C05352=1012.608,-74.665,-110.262,-31.652,71.658,-31.878
C05353=1012.607,-74.904,-110.243,-31.675,71.735,-31.896
C05354=1012.606,-75.144,-110.222,-31.698,71.811,-31.914
C05355=1012.605,-75.384,-110.202,-31.722,71.889,-31.932
C05356=1012.604,-75.624,-110.182,-31.745,71.965,-31.950
C05357=1012.603,-75.953,-110.153,-31.778,72.071,-31.977
C05358=1012.600,-76.343,-110.120,-31.818,72.198,-32.009
C05359=1012.601,-76.583,-110.100,-31.843,72.276,-32.028
C05360=1012.599,-76.822,-110.079,-31.869,72.354,-32.050
C05361=1012.598,-77.061,-110.059,-31.894,72.432,-32.070
C05362=1012.597,-77.300,-110.039,-31.920,72.510,-32.092
C05363=1012.596,-77.540,-110.019,-31.946,72.590,-32.112
C05364=1012.595,-77.779,-109.998,-31.973,72.668,-32.135
C05365=1012.594,-78.018,-109.978,-31.999,72.748,-32.156
C05366=1012.593,-78.257,-109.957,-32.027,72.828,-32.179
C05367=1012.593,-78.496,-109.937,-32.054,72.907,-32.201
C05368=1012.591,-78.734,-109.917,-32.082,72.987,-32.225
C05369=1012.591,-78.972,-109.897,-32.111,73.067,-32.250
C05370=1012.590,-79.211,-109.876,-32.140,73.147,-32.274
C05371=1012.588,-79.449,-109.856,-32.168,73.228,-32.298
C05372=1012.588,-79.687,-109.836,-32.198,73.307,-32.323
C05373=1012.587,-79.925,-109.816,-32.228,73.389,-32.349
C05374=1012.586,-80.163,-109.795,-32.257,73.470,-32.373
C05375=1012.585,-80.400,-109.775,-32.288,73.551,-32.400
C05376=1012.584,-80.637,-109.755,-32.318,73.632,-32.425
C05377=1012.583,-80.874,-109.735,-32.350,73.713,-32.453
C05378=1012.582,-81.111,-109.715,-32.382,73.795,-32.481
C05379=1012.581,-81.347,-109.694,-32.414,73.876,-32.509
C05380=1012.581,-81.583,-109.674,-32.446,73.958,-32.536
C05381=1012.579,-81.820,-109.654,-32.480,74.040,-32.567
C05382=1012.578,-82.058,-109.634,-32.514,74.123,-32.596
C05383=1012.578,-82.294,-109.614,-32.548,74.206,-32.626
C05384=1012.577,-82.532,-109.593,-32.582,74.288,-32.655
C05385=1012.576,-82.766,-109.574,-32.617,74.371,-32.686
C05386=1012.575,-83.003,-109.554,-32.651,74.454,-32.716
C05387=1012.574,-83.239,-109.533,-32.688,74.538,-32.750
C05388=1012.574,-83.475,-109.513,-32.724,74.621,-32.780
///RCONF 0,0,0,0,0,0,0,0,0,0,0,0,0,0,0,0,0,0,0,0,0,0,0,0
C05389=1012.572,-83.710,-109.494,-32.762,74.705,-32.815
C05390=1012.571,-83.943,-109.473,-32.799,74.787,-32.849
C05391=1012.570,-84.175,-109.454,-32.835,74.870,-32.879
C05392=1012.570,-84.409,-109.434,-32.874,74.953,-32.916
C05393=1012.568,-84.649,-109.413,-32.913,75.039,-32.951
C05394=1012.568,-84.904,-109.392,-32.956,75.132,-32.989
C05395=1012.568,-85.180,-109.368,-33.004,75.230,-33.034
C05396=1012.566,-85.465,-109.344,-33.054,75.334,-33.079
C05397=1012.565,-85.747,-109.320,-33.103,75.436,-33.124
C05398=1012.564,-86.017,-109.297,-33.153,75.535,-33.169
C05399=1012.563,-86.268,-109.276,-33.199,75.626,-33.211
C05400=1012.561,-86.502,-109.256,-33.242,75.712,-33.251
C05401=1012.561,-86.733,-109.236,-33.285,75.796,-33.290
C05402=1012.560,-86.963,-109.217,-33.331,75.881,-33.334
C05403=1012.560,-87.186,-109.198,-33.374,75.962,-33.374
C05404=1012.559,-87.405,-109.179,-33.418,76.044,-33.414
C05405=1012.558,-87.624,-109.160,-33.463,76.125,-33.455
C05406=1012.558,-87.840,-109.142,-33.506,76.204,-33.495
C05407=1012.556,-88.056,-109.123,-33.551,76.286,-33.538
C05408=1012.556,-88.282,-109.104,-33.600,76.369,-33.583
C05409=1012.555,-88.509,-109.084,-33.648,76.454,-33.628
C05410=1012.554,-88.742,-109.065,-33.700,76.541,-33.677
C05411=1012.553,-89.009,-109.042,-33.757,76.642,-33.730
C05412=1012.552,-89.306,-109.017,-33.825,76.753,-33.795
C05413=1012.552,-89.614,-108.991,-33.895,76.869,-33.860
C05414=1012.550,-89.915,-108.965,-33.967,76.983,-33.929
C05415=1012.549,-90.193,-108.942,-34.035,77.088,-33.993
C05416=1012.548,-90.433,-108.920,-34.094,77.180,-34.050
C05417=1012.547,-90.854,-108.885,-34.200,77.340,-34.150
C05418=1012.546,-91.137,-108.861,-34.274,77.448,-34.222
C05419=1012.545,-91.368,-108.841,-34.333,77.537,-34.278
C05420=1012.544,-91.600,-108.822,-34.396,77.626,-34.338
C05421=1012.543,-91.830,-108.802,-34.460,77.715,-34.400
C05422=1012.542,-92.061,-108.782,-34.525,77.804,-34.462
C05423=1012.542,-92.293,-108.763,-34.590,77.894,-34.525
C05424=1012.541,-92.523,-108.743,-34.657,77.983,-34.589
C05425=1012.541,-92.753,-108.723,-34.724,78.072,-34.654
C05426=1012.540,-92.983,-108.703,-34.792,78.162,-34.719
C05427=1012.539,-93.213,-108.683,-34.862,78.251,-34.787
C05428=1012.538,-93.443,-108.664,-34.935,78.341,-34.858
C05429=1012.538,-93.672,-108.645,-35.006,78.431,-34.927
C05430=1012.537,-93.901,-108.625,-35.080,78.520,-34.999
C05431=1012.536,-94.129,-108.606,-35.156,78.611,-35.072
C05432=1012.535,-94.357,-108.586,-35.232,78.700,-35.147
C05433=1012.535,-94.584,-108.567,-35.310,78.790,-35.223
C05434=1012.535,-94.811,-108.547,-35.388,78.880,-35.299
C05435=1012.534,-95.038,-108.529,-35.467,78.969,-35.376
C05436=1012.533,-95.265,-108.509,-35.551,79.059,-35.458
C05437=1012.532,-95.490,-108.490,-35.633,79.148,-35.538
C05438=1012.531,-95.716,-108.471,-35.719,79.238,-35.623
C05439=1012.530,-95.941,-108.451,-35.804,79.328,-35.706
C05440=1012.530,-96.166,-108.432,-35.893,79.418,-35.793
C05441=1012.530,-96.390,-108.413,-35.984,79.508,-35.883
C05442=1012.529,-96.614,-108.394,-36.074,79.597,-35.971
C05443=1012.528,-96.839,-108.375,-36.167,79.688,-36.062
C05444=1012.528,-97.063,-108.356,-36.263,79.777,-36.157
C05445=1012.527,-97.286,-108.337,-36.359,79.868,-36.252
C05446=1012.527,-97.510,-108.318,-36.459,79.958,-36.350
C05447=1012.526,-97.733,-108.299,-36.559,80.048,-36.449
C05448=1012.525,-97.957,-108.280,-36.662,80.139,-36.550
C05449=1012.525,-98.180,-108.261,-36.768,80.230,-36.656
C05450=1012.524,-98.405,-108.242,-36.875,80.320,-36.761
C05451=1012.524,-98.628,-108.223,-36.986,80.411,-36.872
C05452=1012.523,-98.852,-108.204,-37.099,80.503,-36.983
C05453=1012.522,-99.076,-108.185,-37.214,80.594,-37.097
C05454=1012.521,-99.300,-108.165,-37.332,80.685,-37.214
C05455=1012.521,-99.524,-108.146,-37.453,80.778,-37.334
C05456=1012.521,-99.749,-108.127,-37.575,80.869,-37.456
C05457=1012.520,-99.975,-108.108,-37.703,80.961,-37.583
C05458=1012.519,-100.200,-108.089,-37.833,81.054,-37.711
C05459=1012.518,-100.426,-108.070,-37.968,81.147,-37.846
C05460=1012.518,-100.652,-108.050,-38.106,81.241,-37.984
C05461=1012.517,-100.879,-108.032,-38.243,81.334,-38.120
C05462=1012.517,-101.106,-108.012,-38.390,81.428,-38.267
C05463=1012.517,-101.333,-107.993,-38.537,81.522,-38.413
C05464=1012.516,-101.561,-107.973,-38.691,81.616,-38.567
C05465=1012.515,-101.789,-107.954,-38.844,81.711,-38.718
C05466=1012.515,-102.018,-107.934,-39.008,81.806,-38.883
C05467=1012.515,-102.247,-107.915,-39.171,81.901,-39.046
C05468=1012.514,-102.476,-107.895,-39.339,81.996,-39.214
C05469=1012.513,-102.705,-107.876,-39.515,82.091,-39.389
C05470=1012.513,-102.934,-107.856,-39.694,82.188,-39.568
C05471=1012.513,-103.164,-107.837,-39.878,82.283,-39.753
C05472=1012.512,-103.394,-107.817,-40.070,82.379,-39.945
C05473=1012.512,-103.624,-107.797,-40.264,82.475,-40.138
C05474=1012.511,-103.940,-107.770,-40.542,82.608,-40.416
C05475=1012.510,-104.316,-107.739,-40.887,82.765,-40.762
C05476=1012.509,-104.546,-107.719,-41.106,82.862,-40.981
C05477=1012.509,-104.777,-107.699,-41.335,82.959,-41.211
C05478=1012.509,-105.008,-107.680,-41.567,83.055,-41.443
C05479=1012.508,-105.240,-107.660,-41.809,83.153,-41.685
C05480=1012.507,-105.471,-107.641,-42.059,83.250,-41.936
C05481=1012.507,-105.703,-107.621,-42.315,83.347,-42.193
C05482=1012.507,-105.934,-107.602,-42.580,83.445,-42.458
C05483=1012.506,-106.166,-107.581,-42.857,83.542,-42.736
C05484=1012.507,-106.400,-107.561,-43.142,83.641,-43.022
C05485=1012.505,-106.643,-107.541,-43.453,83.743,-43.334
C05486=1012.505,-106.896,-107.519,-43.783,83.849,-43.664
C05487=1012.505,-107.158,-107.497,-44.142,83.959,-44.025
C05488=1012.505,-107.428,-107.474,-44.528,84.074,-44.412
C05489=1012.504,-107.703,-107.451,-44.934,84.189,-44.819
C05490=1012.503,-107.980,-107.427,-45.362,84.305,-45.249
C05491=1012.503,-108.254,-107.404,-45.802,84.419,-45.692
C05492=1012.503,-108.523,-107.381,-46.257,84.532,-46.148
C05493=1012.503,-108.783,-107.359,-46.709,84.640,-46.601
C05494=1012.502,-109.033,-107.338,-47.169,84.745,-47.062
C05495=1012.502,-109.274,-107.318,-47.630,84.845,-47.525
C05496=1012.501,-109.507,-107.298,-48.097,84.942,-47.994
C05497=1012.501,-109.739,-107.278,-48.576,85.038,-48.475
C05498=1012.501,-109.970,-107.259,-49.075,85.134,-48.976
C05499=1012.501,-110.202,-107.239,-49.594,85.228,-49.497
C05500=1012.500,-110.434,-107.219,-50.135,85.324,-50.039
C05501=1012.500,-110.665,-107.199,-50.705,85.419,-50.612
C05502=1012.500,-110.897,-107.180,-51.293,85.513,-51.202
C05503=1012.499,-111.128,-107.160,-51.914,85.607,-51.825
C05504=1012.499,-111.359,-107.140,-52.563,85.700,-52.476
C05505=1012.499,-111.590,-107.121,-53.233,85.794,-53.148
C05506=1012.499,-111.822,-107.101,-53.942,85.886,-53.860
C05507=1012.498,-112.053,-107.082,-54.684,85.978,-54.605
C05508=1012.498,-112.284,-107.062,-55.462,86.070,-55.385
C05509=1012.499,-112.516,-107.042,-56.287,86.161,-56.212
C05510=1012.498,-112.748,-107.023,-57.142,86.251,-57.070
C05511=1012.498,-112.979,-107.003,-58.042,86.340,-57.972
C05512=1012.497,-113.210,-106.984,-58.994,86.429,-58.928
C05513=1012.498,-113.441,-106.964,-59.988,86.516,-59.924
C05514=1012.498,-113.672,-106.945,-61.044,86.603,-60.983
C05515=1012.498,-113.903,-106.925,-62.143,86.688,-62.085
C05516=1012.498,-114.135,-106.905,-63.313,86.772,-63.258
C05517=1012.497,-114.366,-106.886,-64.545,86.855,-64.493
C05518=1012.497,-114.598,-106.866,-65.843,86.936,-65.795
C05519=1012.496,-114.829,-106.846,-67.217,87.016,-67.172
C05520=1012.497,-115.061,-106.827,-68.666,87.095,-68.624
C05521=1012.497,-115.272,-106.810,-70.066,87.164,-70.028
C05522=1012.497,-115.485,-106.791,-71.544,87.233,-71.508
C05523=1012.497,-115.754,-106.768,-73.538,87.317,-73.507
C05524=1012.496,-115.985,-106.749,-75.331,87.386,-75.303
C05525=1012.496,-116.217,-106.729,-77.246,87.453,-77.222
C05526=1012.496,-116.447,-106.710,-79.234,87.516,-79.213
C05527=1012.496,-116.679,-106.690,-81.352,87.577,-81.336
C05528=1012.496,-116.910,-106.670,-83.577,87.635,-83.564
C05529=1012.496,-117.141,-106.651,-85.907,87.688,-85.899
C05530=1012.497,-117.373,-106.632,-88.359,87.738,-88.354
C05531=1012.497,-117.604,-106.612,-90.919,87.783,-90.919
C05532=1012.496,-117.835,-106.593,-93.576,87.824,-93.580
C05533=1012.497,-118.066,-106.573,-96.329,87.860,-96.336
C05534=1012.496,-118.297,-106.554,-99.188,87.891,-99.200
C05535=1012.496,-118.529,-106.534,-102.102,87.916,-102.119
C05536=1012.497,-118.759,-106.514,-105.100,87.936,-105.121
C05537=1012.496,-118.990,-106.495,-108.145,87.950,-108.171
C05538=1012.496,-119.222,-106.475,-111.225,87.958,-111.255
C05539=1012.497,-119.453,-106.456,-114.338,87.960,-114.373
C05540=1012.497,-119.684,-106.437,-117.448,87.956,-117.488
C05541=1012.497,-119.916,-106.417,-120.535,87.946,-120.579
C05542=1012.498,-120.147,-106.397,-123.598,87.930,-123.648
C05543=1012.497,-120.378,-106.378,-126.611,87.908,-126.666
C05544=1012.498,-120.608,-106.359,-129.528,87.881,-129.588
C05545=1012.498,-120.840,-106.339,-132.400,87.848,-132.465
C05546=1012.498,-121.070,-106.320,-135.162,87.810,-135.232
C05547=1012.498,-121.302,-106.300,-137.833,87.766,-137.910
C05548=1012.499,-121.533,-106.281,-140.407,87.718,-140.488
C05549=1012.498,-121.764,-106.262,-142.856,87.666,-142.943
C05550=1012.498,-121.996,-106.242,-145.213,87.609,-145.305
C05551=1012.499,-122.227,-106.222,-147.454,87.548,-147.552
C05552=1012.499,-122.457,-106.203,-149.582,87.484,-149.685
C05553=1012.499,-122.689,-106.184,-151.598,87.416,-151.707
C05554=1012.500,-122.920,-106.164,-153.513,87.344,-153.629
C05555=1012.499,-123.151,-106.145,-155.336,87.270,-155.458
C05556=1012.500,-123.382,-106.125,-157.042,87.194,-157.170
C05557=1012.500,-123.613,-106.105,-158.676,87.115,-158.810
C05558=1012.501,-123.844,-106.086,-160.231,87.033,-160.370
C05559=1012.500,-124.076,-106.067,-161.687,86.949,-161.833
C05560=1012.501,-124.306,-106.048,-163.063,86.863,-163.216
C05561=1012.502,-124.537,-106.028,-164.377,86.775,-164.537
C05562=1012.501,-124.768,-106.009,-165.619,86.686,-165.785
C05563=1012.502,-124.999,-105.989,-166.793,86.595,-166.966
C05564=1012.502,-125.230,-105.970,-167.904,86.502,-168.083
C05565=1012.503,-125.462,-105.950,-168.968,86.408,-169.154
C05566=1012.503,-125.692,-105.931,-169.965,86.313,-170.158
C05567=1012.503,-125.923,-105.912,-170.920,86.216,-171.120
C05568=1012.503,-126.155,-105.892,-171.826,86.118,-172.033
C05569=1012.504,-126.464,-105.867,-172.966,85.987,-173.183
C05570=1012.504,-126.848,-105.834,-174.287,85.819,-174.516
C05571=1012.505,-127.079,-105.815,-175.034,85.718,-175.270
C05572=1012.506,-127.309,-105.795,-175.744,85.615,-175.989
C05573=1012.507,-127.541,-105.776,-176.421,85.512,-176.672
C05574=1012.506,-127.772,-105.757,-177.074,85.407,-177.333
C05575=1012.507,-128.003,-105.737,-177.688,85.303,-177.955
C05576=1012.508,-128.233,-105.718,-178.282,85.198,-178.556
C05577=1012.509,-128.465,-105.699,-178.849,85.091,-179.131
C05578=1012.509,-128.695,-105.679,-179.390,84.985,-179.681
C05579=1012.509,-128.927,-105.660,-179.915,84.877,179.787
C05580=1012.509,-129.157,-105.640,179.584,84.768,179.277
C05581=1012.510,-129.389,-105.622,179.110,84.661,178.795
C05582=1012.511,-129.619,-105.602,178.644,84.551,178.321
C05583=1012.512,-129.850,-105.582,178.204,84.442,177.873
C05584=1012.513,-130.082,-105.564,177.783,84.332,177.442
C05585=1012.513,-130.312,-105.544,177.372,84.221,177.023
C05586=1012.513,-130.543,-105.525,176.979,84.110,176.621
C05587=1012.513,-130.774,-105.505,176.601,83.999,176.234
C05588=1012.514,-131.006,-105.486,176.233,83.886,175.858
C05589=1012.515,-131.236,-105.467,175.884,83.774,175.500
C05590=1012.516,-131.467,-105.447,175.545,83.661,175.151
C05591=1012.517,-131.698,-105.428,175.217,83.549,174.814
C05592=1012.517,-131.929,-105.409,174.903,83.435,174.491
C05593=1012.518,-132.160,-105.389,174.595,83.321,174.174
C05594=1012.518,-132.391,-105.371,174.299,83.207,173.869
C05595=1012.519,-132.622,-105.351,174.019,83.093,173.578
C05596=1012.520,-132.852,-105.332,173.739,82.978,173.290
C05597=1012.521,-133.084,-105.313,173.474,82.863,173.015
C05598=1012.521,-133.315,-105.293,173.220,82.747,172.750
C05599=1012.522,-133.545,-105.274,172.970,82.632,172.490
C05600=1012.523,-133.777,-105.255,172.728,82.516,172.238
C05601=1012.524,-134.007,-105.235,172.495,82.399,171.996
C05602=1012.845,-81.888,-107.547,164.895,61.170,160.790
C05603=1012.843,-81.675,-107.564,164.893,61.240,160.803
C05604=1012.841,-81.438,-107.584,164.892,61.318,160.818
C05605=1012.839,-81.201,-107.604,164.889,61.395,160.832
C05606=1012.837,-80.965,-107.625,164.887,61.471,160.846
C05607=1012.835,-80.729,-107.644,164.885,61.548,160.861
C05608=1012.834,-80.492,-107.664,164.883,61.625,160.875
C05609=1012.832,-80.255,-107.684,164.880,61.701,160.889
C05610=1012.830,-80.018,-107.704,164.880,61.777,160.904
C05611=1012.828,-79.779,-107.724,164.877,61.853,160.918
C05612=1012.827,-79.542,-107.744,164.875,61.929,160.933
C05613=1012.824,-79.303,-107.764,164.874,62.005,160.947
C05614=1012.823,-79.065,-107.784,164.872,62.081,160.962
C05615=1012.821,-78.827,-107.803,164.871,62.155,160.976
C05616=1012.819,-78.588,-107.823,164.870,62.230,160.991
C05617=1012.818,-78.349,-107.843,164.869,62.305,161.005
C05618=1012.816,-78.110,-107.864,164.867,62.380,161.019
C05619=1012.814,-77.871,-107.884,164.866,62.454,161.034
C05620=1012.813,-77.632,-107.904,164.865,62.528,161.048
C05621=1012.812,-77.393,-107.924,164.865,62.602,161.063
C05622=1012.809,-77.154,-107.944,164.863,62.676,161.077
C05623=1012.808,-76.914,-107.964,164.863,62.749,161.092
C05624=1012.807,-76.675,-107.984,164.861,62.822,161.106
C05625=1012.805,-76.435,-108.004,164.861,62.895,161.121
C05626=1012.803,-76.196,-108.025,164.860,62.968,161.135
C05627=1012.801,-75.956,-108.045,164.860,63.040,161.150
C05628=1012.800,-75.716,-108.065,164.859,63.112,161.164
C05629=1012.799,-75.476,-108.084,164.860,63.185,161.179
C05630=1012.797,-75.237,-108.105,164.859,63.256,161.193
C05631=1012.796,-74.996,-108.125,164.860,63.328,161.208
C05632=1012.794,-74.756,-108.145,164.859,63.399,161.222
C05633=1012.792,-74.517,-108.166,164.859,63.470,161.237
C05634=1012.791,-74.276,-108.186,164.859,63.541,161.251
C05635=1012.789,-74.036,-108.206,164.860,63.612,161.266
C05636=1012.788,-73.796,-108.227,164.860,63.681,161.280
C05637=1012.786,-73.556,-108.247,164.861,63.751,161.295
C05638=1012.785,-73.315,-108.267,164.860,63.821,161.309
C05639=1012.783,-73.075,-108.287,164.861,63.891,161.324
C05640=1012.782,-72.834,-108.307,164.862,63.960,161.338
C05641=1012.781,-72.594,-108.328,164.863,64.028,161.353
C05642=1012.779,-72.354,-108.348,164.864,64.098,161.368
C05643=1012.778,-72.113,-108.368,164.864,64.166,161.382
C05644=1012.776,-71.873,-108.388,164.865,64.235,161.396
C05645=1012.774,-71.633,-108.408,164.867,64.302,161.411
C05646=1012.773,-71.392,-108.428,164.868,64.370,161.426
C05647=1012.772,-71.151,-108.448,164.869,64.438,161.440
C05648=1012.771,-70.910,-108.469,164.870,64.505,161.454
C05649=1012.769,-70.670,-108.489,164.871,64.572,161.469
C05650=1012.768,-70.429,-108.509,164.873,64.639,161.483
C05651=1012.766,-70.188,-108.530,164.875,64.704,161.498
C05652=1012.765,-69.947,-108.550,164.875,64.771,161.512
C05653=1012.763,-69.706,-108.570,164.878,64.837,161.527
C05654=1012.762,-69.465,-108.591,164.879,64.902,161.541
C05655=1012.761,-69.225,-108.611,164.882,64.968,161.556
C05656=1012.760,-68.984,-108.631,164.883,65.032,161.570
C05657=1012.758,-68.743,-108.651,164.885,65.097,161.585
C05658=1012.757,-68.502,-108.671,164.886,65.162,161.599
C05659=1012.756,-68.262,-108.692,164.888,65.226,161.613
C05660=1012.754,-68.021,-108.712,164.891,65.290,161.628
C05661=1012.753,-67.780,-108.732,164.894,65.354,161.643
C05662=1012.752,-67.539,-108.752,164.896,65.417,161.657
C05663=1012.750,-67.299,-108.773,164.898,65.481,161.672
C05664=1012.749,-67.058,-108.793,164.900,65.543,161.686
C05665=1012.748,-66.818,-108.814,164.903,65.606,161.700
C05666=1012.746,-66.578,-108.834,164.905,65.668,161.714
C05667=1012.745,-66.337,-108.854,164.908,65.731,161.729
C05668=1012.744,-66.097,-108.875,164.910,65.792,161.743
C05669=1012.743,-65.856,-108.894,164.913,65.854,161.757
C05670=1012.742,-65.616,-108.914,164.916,65.915,161.772
C05671=1012.741,-65.376,-108.935,164.918,65.976,161.786
C05672=1012.739,-65.136,-108.955,164.921,66.036,161.800
C05673=1012.737,-64.754,-108.987,164.926,66.132,161.823
C05674=1012.736,-64.417,-109.015,164.931,66.216,161.843
C05675=1012.734,-64.178,-109.036,164.934,66.276,161.858
C05676=1012.734,-63.938,-109.056,164.938,66.335,161.872
C05677=1012.732,-63.699,-109.077,164.941,66.394,161.886
C05678=1012.731,-63.459,-109.097,164.943,66.453,161.900
C05679=1012.730,-63.221,-109.116,164.948,66.511,161.915
C05680=1012.729,-62.982,-109.136,164.951,66.569,161.929
C05681=1012.728,-62.743,-109.157,164.953,66.627,161.943
C05682=1012.726,-62.505,-109.177,164.958,66.684,161.957
C05683=1012.725,-62.266,-109.197,164.962,66.741,161.971
C05684=1012.724,-62.028,-109.217,164.965,66.798,161.985
C05685=1012.723,-61.790,-109.237,164.969,66.855,161.999
C05686=1012.723,-61.552,-109.257,164.973,66.911,162.014
C05687=1012.722,-61.314,-109.277,164.977,66.967,162.028
C05688=1012.720,-61.077,-109.297,164.980,67.023,162.041
C05689=1012.719,-60.840,-109.317,164.984,67.078,162.056
C05690=1012.718,-60.603,-109.337,164.987,67.133,162.069
C05691=1012.717,-60.365,-109.356,164.992,67.187,162.083
C05692=1012.716,-60.129,-109.377,164.996,67.242,162.097
C05693=1012.715,-59.892,-109.396,165.001,67.296,162.111
C05694=1012.714,-59.656,-109.417,165.005,67.350,162.125
C05695=1012.713,-59.420,-109.437,165.009,67.403,162.139
C05696=1012.712,-59.183,-109.457,165.013,67.457,162.153
C05697=1012.710,-58.948,-109.476,165.018,67.510,162.167
C05698=1012.710,-58.711,-109.496,165.022,67.562,162.181
C05699=1012.710,-58.477,-109.516,165.027,67.615,162.195
C05700=1012.708,-58.242,-109.536,165.031,67.666,162.208
C05701=1012.707,-58.006,-109.556,165.036,67.719,162.222
C05702=1012.706,-57.771,-109.576,165.040,67.770,162.236
C05703=1012.705,-57.536,-109.595,165.045,67.821,162.250
C05704=1012.704,-57.302,-109.615,165.049,67.872,162.263
C05705=1012.704,-57.068,-109.635,165.053,67.923,162.276
C05706=1012.702,-56.833,-109.654,165.058,67.973,162.290
C05707=1012.701,-56.599,-109.674,165.063,68.023,162.304
C05708=1012.701,-56.365,-109.694,165.069,68.073,162.318
C05709=1012.699,-56.131,-109.714,165.073,68.123,162.331
C05710=1012.698,-55.897,-109.733,165.078,68.172,162.345
C05711=1012.697,-55.663,-109.753,165.084,68.221,162.358
C05712=1012.697,-55.429,-109.773,165.088,68.269,162.371
C05713=1012.697,-55.196,-109.793,165.092,68.318,162.385
C05714=1012.695,-54.962,-109.813,165.098,68.367,162.399
C05715=1012.694,-54.728,-109.832,165.103,68.414,162.412
C05716=1012.693,-54.494,-109.852,165.108,68.463,162.425
C05717=1012.693,-54.261,-109.871,165.113,68.510,162.438
C05718=1012.692,-54.027,-109.891,165.118,68.557,162.452
C05719=1012.691,-53.794,-109.911,165.123,68.604,162.465
C05720=1012.690,-53.560,-109.930,165.128,68.651,162.479
C05721=1012.689,-53.326,-109.950,165.134,68.697,162.492
C05722=1012.688,-53.092,-109.970,165.139,68.745,162.505
C05723=1012.687,-52.858,-109.989,165.145,68.791,162.519
C05724=1012.686,-52.625,-110.009,165.150,68.836,162.532
C05725=1012.686,-52.392,-110.029,165.156,68.882,162.545
C05726=1012.685,-52.157,-110.049,165.161,68.927,162.558
C05727=1012.685,-51.923,-110.068,165.166,68.972,162.571
C05728=1012.683,-51.689,-110.088,165.172,69.017,162.584
C05729=1012.682,-51.456,-110.108,165.177,69.062,162.598
C05730=1012.681,-51.222,-110.127,165.182,69.106,162.610
C05731=1012.681,-50.989,-110.147,165.189,69.151,162.624
C05732=1012.680,-50.755,-110.167,165.194,69.195,162.637
C05733=1012.680,-50.521,-110.187,165.200,69.237,162.650
C05734=1012.679,-50.287,-110.206,165.206,69.281,162.663
C05735=1012.678,-50.053,-110.226,165.212,69.324,162.676
C05736=1012.677,-49.819,-110.245,165.217,69.368,162.689
C05737=1012.677,-49.586,-110.265,165.222,69.410,162.702
C05738=1012.675,-49.352,-110.285,165.228,69.453,162.715
C05739=1012.675,-49.118,-110.305,165.235,69.496,162.728
C05740=1012.674,-48.884,-110.325,165.241,69.537,162.741
C05741=1012.673,-48.650,-110.344,165.246,69.579,162.754
C05742=1012.672,-48.416,-110.364,165.253,69.620,162.767
C05743=1012.672,-48.183,-110.383,165.259,69.662,162.780
C05744=1012.672,-47.949,-110.404,165.265,69.703,162.792
C05745=1012.671,-47.715,-110.423,165.270,69.743,162.805
C05746=1012.670,-47.481,-110.442,165.276,69.784,162.817
C05747=1012.669,-47.248,-110.462,165.281,69.825,162.830
C05748=1012.669,-47.013,-110.482,165.288,69.865,162.843
C05749=1012.667,-46.779,-110.502,165.294,69.904,162.856
C05750=1012.666,-46.545,-110.521,165.300,69.944,162.868
C05751=1012.666,-46.312,-110.541,165.306,69.983,162.881
C05752=1012.666,-46.078,-110.561,165.312,70.023,162.893
C05753=1012.665,-45.844,-110.581,165.319,70.062,162.906
C05754=1012.664,-45.610,-110.600,165.325,70.100,162.918
C05755=1012.664,-45.376,-110.620,165.330,70.139,162.930
C05756=1012.663,-45.142,-110.640,165.336,70.177,162.943
C05757=1012.662,-44.908,-110.659,165.343,70.215,162.955
C05758=1012.662,-44.674,-110.679,165.348,70.253,162.967
C05759=1012.661,-44.440,-110.698,165.356,70.290,162.980
C05760=1012.661,-44.206,-110.718,165.362,70.328,162.992
C05761=1012.659,-43.972,-110.739,165.368,70.365,163.005
C05762=1012.659,-43.739,-110.758,165.375,70.402,163.017
C05763=1012.658,-43.504,-110.778,165.380,70.438,163.029
C05764=1012.658,-43.270,-110.798,165.385,70.474,163.040
C05765=1012.657,-43.036,-110.817,165.394,70.511,163.054
C05766=1012.656,-42.802,-110.837,165.400,70.547,163.065
C05767=1012.656,-42.569,-110.856,165.406,70.582,163.077
C05768=1012.655,-42.334,-110.876,165.412,70.618,163.089
C05769=1012.655,-42.100,-110.896,165.418,70.653,163.101
C05770=1012.654,-41.866,-110.916,165.424,70.687,163.113
C05771=1012.653,-41.632,-110.935,165.430,70.722,163.124
C05772=1012.653,-41.397,-110.955,165.437,70.756,163.137
C05773=1012.652,-41.164,-110.975,165.444,70.791,163.149
C05774=1012.651,-40.929,-110.995,165.450,70.825,163.160
C05775=1012.651,-40.695,-111.014,165.456,70.858,163.172
C05776=1012.650,-40.461,-111.034,165.461,70.892,163.183
C05777=1012.650,-40.227,-111.054,165.469,70.925,163.195
C05778=1012.649,-39.993,-111.073,165.476,70.959,163.207
C05779=1012.649,-39.758,-111.093,165.481,70.992,163.218
C05780=1012.647,-39.380,-111.125,165.492,71.044,163.237
C05781=1012.647,-39.056,-111.152,165.500,71.089,163.252
C05782=1012.646,-38.822,-111.172,165.506,71.121,163.264
C05783=1012.646,-38.587,-111.192,165.512,71.152,163.275
C05784=1012.645,-38.353,-111.212,165.520,71.184,163.287
C05785=1012.645,-38.119,-111.231,165.526,71.216,163.298
C05786=1012.644,-37.885,-111.251,165.533,71.246,163.309
C05787=1012.644,-37.651,-111.271,165.538,71.277,163.320
C05788=1012.644,-37.416,-111.291,165.545,71.307,163.331
C05789=1012.643,-37.183,-111.310,165.551,71.338,163.342
C05790=1012.642,-36.948,-111.330,165.557,71.368,163.353
C05791=1012.642,-36.714,-111.350,165.563,71.398,163.363
C05792=1012.641,-36.480,-111.369,165.570,71.427,163.375
C05793=1012.640,-36.245,-111.390,165.577,71.457,163.386
C05794=1012.640,-36.011,-111.409,165.583,71.486,163.396
C05795=1012.639,-35.777,-111.429,165.589,71.515,163.407
C05796=1012.639,-35.543,-111.449,165.595,71.543,163.417
C05797=1012.639,-35.308,-111.468,165.601,71.572,163.428
C05798=1012.638,-35.074,-111.487,165.608,71.600,163.439
C05799=1012.637,-34.839,-111.507,165.613,71.629,163.449
C05800=1012.637,-34.605,-111.527,165.620,71.657,163.460
C05801=1012.636,-34.371,-111.546,165.626,71.684,163.470
C05802=1012.636,-34.137,-111.566,165.632,71.712,163.481
C05803=1012.636,-33.902,-111.586,165.638,71.738,163.491
C05804=1012.635,-33.668,-111.606,165.644,71.765,163.501
C05805=1012.635,-33.434,-111.625,165.650,71.791,163.511
C05806=1012.635,-33.200,-111.645,165.657,71.819,163.522
C05807=1012.634,-32.965,-111.666,165.663,71.845,163.532
C05808=1012.633,-32.731,-111.685,165.668,71.871,163.541
C05809=1012.632,-32.497,-111.705,165.674,71.897,163.551
C05810=1012.632,-32.262,-111.725,165.681,71.922,163.562
C05811=1012.631,-32.028,-111.744,165.686,71.948,163.571
C05812=1012.631,-31.794,-111.764,165.693,71.972,163.581
C05813=1012.631,-31.560,-111.784,165.699,71.997,163.591
C05814=1012.631,-31.325,-111.804,165.705,72.022,163.600
C05815=1012.630,-31.091,-111.823,165.710,72.046,163.609
C05816=1012.630,-30.857,-111.843,165.716,72.071,163.619
C05817=1012.629,-30.622,-111.863,165.723,72.094,163.629
C05818=1012.629,-30.389,-111.882,165.728,72.118,163.638
C05819=1012.628,-30.154,-111.902,165.734,72.142,163.647
C05820=1012.628,-29.920,-111.922,165.740,72.165,163.657
C05821=1012.628,-29.685,-111.942,165.745,72.188,163.666
C05822=1012.627,-29.452,-111.961,165.751,72.211,163.675
C05823=1012.627,-29.217,-111.981,165.758,72.234,163.684
C05824=1012.626,-28.982,-112.000,165.763,72.256,163.693
C05825=1012.625,-28.748,-112.020,165.769,72.278,163.702
C05826=1012.625,-28.514,-112.040,165.775,72.300,163.712
C05827=1012.625,-28.279,-112.059,165.780,72.322,163.720
C05828=1012.625,-28.045,-112.079,165.785,72.343,163.728
C05829=1012.624,-27.811,-112.099,165.792,72.365,163.738
C05830=1012.624,-27.577,-112.119,165.798,72.386,163.747
C05831=1012.623,-27.342,-112.138,165.801,72.407,163.754
C05832=1012.622,-27.109,-112.158,165.808,72.427,163.763
C05833=1012.622,-26.874,-112.178,165.813,72.447,163.771
C05834=1012.622,-26.640,-112.198,165.819,72.468,163.780
C05835=1012.621,-26.407,-112.218,165.824,72.488,163.788
C05836=1012.621,-26.172,-112.238,165.829,72.508,163.796
C05837=1012.621,-25.938,-112.257,165.835,72.527,163.805
C05838=1012.621,-25.703,-112.277,165.840,72.546,163.812
C05839=1012.620,-25.469,-112.297,165.845,72.566,163.820
C05840=1012.620,-25.235,-112.317,165.851,72.584,163.829
C05841=1012.619,-25.001,-112.336,165.856,72.603,163.836
C05842=1012.619,-24.767,-112.355,165.860,72.621,163.844
C05843=1012.619,-24.533,-112.375,165.865,72.640,163.852
C05844=1012.619,-24.298,-112.395,165.870,72.657,163.859
C05845=1012.618,-24.064,-112.414,165.876,72.675,163.867
C05846=1012.618,-23.830,-112.434,165.881,72.693,163.874
C05847=1012.618,-23.596,-112.454,165.885,72.710,163.882
C05848=1012.617,-23.362,-112.473,165.890,72.727,163.889
C05849=1012.616,-23.127,-112.493,165.895,72.744,163.896
C05850=1012.616,-22.893,-112.513,165.901,72.761,163.904
C05851=1012.615,-22.659,-112.533,165.906,72.777,163.911
C05852=1012.615,-22.425,-112.552,165.909,72.793,163.917
C05853=1012.615,-22.190,-112.572,165.913,72.809,163.924
C05854=1012.615,-21.958,-112.592,165.918,72.825,163.931
C05855=1012.615,-21.723,-112.612,165.924,72.841,163.938
C05856=1012.615,-21.489,-112.632,165.928,72.856,163.945
C05857=1012.614,-21.255,-112.651,165.933,72.871,163.951
C05858=1012.614,-21.020,-112.671,165.939,72.886,163.959
C05859=1012.613,-20.786,-112.691,165.942,72.901,163.965
C05860=1012.612,-20.552,-112.710,165.946,72.916,163.971
C05861=1012.612,-20.318,-112.730,165.950,72.929,163.977
C05862=1012.612,-20.040,-112.753,165.955,72.946,163.984
C05863=1012.612,-19.690,-112.783,165.963,72.967,163.994
C05864=1012.611,-19.430,-112.805,165.967,72.982,164.001
C05865=1012.611,-19.130,-112.830,165.972,72.999,164.008
C05866=1012.611,-18.804,-112.857,165.977,73.016,164.016
C05867=1012.610,-18.472,-112.885,165.984,73.035,164.024
C05868=1012.609,-18.155,-112.911,165.989,73.052,164.032
C05869=1012.610,-17.870,-112.936,165.994,73.066,164.039
C05870=1012.609,-17.623,-112.956,165.997,73.079,164.044
C05871=1012.609,-17.392,-112.976,166.002,73.090,164.050
C05872=1012.609,-17.161,-112.995,166.006,73.102,164.055
C05873=1012.609,-16.927,-113.015,166.008,73.113,164.059
C05874=1012.608,-16.689,-113.035,166.014,73.124,164.065
C05875=1012.608,-16.452,-113.055,166.016,73.135,164.070
C05876=1012.607,-16.217,-113.075,166.020,73.145,164.075
C05877=1012.607,-15.981,-113.094,166.024,73.156,164.080
C05878=1012.606,-15.745,-113.115,166.027,73.166,164.085
C05879=1012.606,-15.509,-113.134,166.030,73.176,164.089
C05880=1012.606,-15.277,-113.154,166.033,73.186,164.094
C05881=1012.605,-15.047,-113.173,166.037,73.195,164.098
C05882=1012.606,-14.820,-113.193,166.040,73.204,164.103
C05883=1012.605,-14.595,-113.211,166.042,73.213,164.106
C05884=1012.605,-14.372,-113.230,166.046,73.222,164.110
C05885=1012.604,-14.149,-113.249,166.049,73.229,164.114
C05886=1012.604,-13.925,-113.267,166.052,73.238,164.119
C05887=1012.604,-13.699,-113.287,166.056,73.246,164.123
C05888=1012.604,-13.470,-113.306,166.059,73.254,164.127
C05889=1012.604,-13.237,-113.326,166.061,73.262,164.130
C05890=1012.604,-13.000,-113.346,166.064,73.270,164.134
C05891=1012.603,-12.759,-113.366,166.067,73.277,164.138
C05892=1012.603,-12.514,-113.386,166.069,73.284,164.141
C05893=1012.603,-12.268,-113.406,166.072,73.292,164.145
C05894=1012.602,-12.021,-113.428,166.075,73.300,164.149
C05895=1012.602,-11.775,-113.448,166.078,73.306,164.152
C05896=1012.602,-11.527,-113.470,166.080,73.313,164.155
C05897=1012.602,-11.279,-113.490,166.083,73.319,164.158
C05898=1012.601,-11.031,-113.511,166.086,73.325,164.162
C05899=1012.602,-10.782,-113.532,166.087,73.332,164.164
C05900=1012.601,-10.532,-113.553,166.092,73.338,164.168
C05901=1012.601,-10.282,-113.574,166.093,73.344,164.171
C05902=1012.600,-10.032,-113.595,166.094,73.349,164.173
C05903=1012.600,-9.781,-113.616,166.097,73.354,164.176
C05904=1012.600,-9.530,-113.637,166.100,73.359,164.179
C05905=1012.600,-9.279,-113.659,166.102,73.364,164.181
C05906=1012.599,-9.028,-113.679,166.105,73.369,164.184
C05907=1012.599,-8.776,-113.700,166.106,73.373,164.186
C05908=1012.599,-8.525,-113.722,166.108,73.376,164.188
C05909=1012.599,-8.274,-113.743,166.109,73.381,164.190
C05910=1012.598,-8.021,-113.764,166.111,73.384,164.192
C05911=1012.598,-7.769,-113.785,166.114,73.388,164.195
C05912=1012.598,-7.516,-113.807,166.116,73.391,164.197
C05913=1012.598,-7.261,-113.828,166.117,73.394,164.198
C05914=1012.597,-7.007,-113.850,166.119,73.396,164.200
C05915=1012.597,-6.750,-113.871,166.119,73.399,164.201
C05916=1012.597,-6.493,-113.892,166.121,73.401,164.203
C05917=1012.597,-6.236,-113.914,166.123,73.403,164.204
C05918=1012.596,-5.977,-113.936,166.125,73.405,164.206
C05919=1012.596,-5.718,-113.958,166.125,73.407,164.207
C05920=1012.596,-5.461,-113.979,166.127,73.407,164.208
C05921=1012.596,-5.204,-114.001,166.127,73.409,164.208
C05922=1012.595,-4.951,-114.022,166.129,73.409,164.209
C05923=1012.596,-4.708,-114.043,166.131,73.410,164.210
C05924=1012.596,-4.472,-114.062,166.131,73.410,164.210
C05925=1012.595,-4.243,-114.081,166.132,73.411,164.212
C05926=1012.595,-4.017,-114.101,166.134,73.410,164.212
C05927=1012.595,-3.791,-114.120,166.134,73.410,164.212
C05928=1012.595,-3.561,-114.139,166.135,73.410,164.213
C05929=1012.595,-3.324,-114.159,166.136,73.409,164.213
C05930=1012.594,-3.081,-114.180,166.136,73.408,164.213
C05931=1012.594,-2.836,-114.201,166.137,73.407,164.213
C05932=1012.594,-2.592,-114.220,166.137,73.406,164.213
C05933=1012.593,-2.348,-114.242,166.136,73.404,164.212
C05934=1012.593,-2.104,-114.262,166.137,73.402,164.212
C05935=1012.593,-1.862,-114.283,166.138,73.400,164.212
C05936=1012.593,-1.619,-114.302,166.138,73.398,164.211
C05937=1012.593,-1.378,-114.323,166.139,73.396,164.211
C05938=1012.593,-1.137,-114.343,166.138,73.393,164.210
C05939=1012.593,-0.897,-114.363,166.139,73.391,164.210
C05940=1012.593,-0.659,-114.383,166.139,73.387,164.209
C05941=1012.592,-0.420,-114.403,166.139,73.385,164.208
C05942=1012.592,-0.181,-114.423,166.138,73.381,164.206
C05943=1012.592,0.055,-114.444,166.138,73.377,164.205
C05944=1012.592,0.291,-114.463,166.139,73.374,164.205
C05945=1012.592,0.526,-114.483,166.138,73.370,164.203
C05946=1012.592,0.760,-114.503,166.137,73.365,164.201
C05947=1012.591,0.995,-114.522,166.136,73.361,164.200
C05948=1012.591,1.231,-114.541,166.136,73.357,164.198
C05949=1012.591,1.468,-114.562,166.136,73.352,164.197
C05950=1012.591,1.705,-114.582,166.137,73.347,164.196
C05951=1012.591,1.939,-114.602,166.135,73.341,164.194
C05952=1012.590,2.169,-114.621,166.136,73.337,164.192
C05953=1012.590,2.389,-114.639,166.133,73.332,164.190
C05954=1012.590,2.798,-114.673,166.132,73.322,164.186
C05955=1012.590,3.182,-114.706,166.133,73.312,164.184
C05956=1012.590,3.574,-114.739,166.130,73.301,164.179
C05957=1012.590,3.781,-114.756,166.129,73.295,164.177
C05958=1012.589,4.001,-114.775,166.129,73.289,164.175
C05959=1012.589,4.229,-114.794,166.127,73.282,164.172
C05960=1012.589,4.462,-114.814,166.127,73.275,164.170
C05961=1012.589,4.695,-114.834,166.125,73.268,164.167
C05962=1012.589,4.927,-114.853,166.125,73.260,164.165
C05963=1012.589,5.158,-114.872,166.124,73.253,164.163
C05964=1012.589,5.390,-114.891,166.122,73.245,164.159
C05965=1012.588,5.622,-114.911,166.120,73.236,164.156
C05966=1012.588,5.855,-114.931,166.120,73.229,164.153
C05967=1012.588,6.089,-114.950,166.118,73.221,164.150
C05968=1012.588,6.324,-114.970,166.117,73.212,164.147
C05969=1012.588,6.557,-114.990,166.115,73.202,164.143
C05970=1012.588,6.790,-115.010,166.113,73.194,164.140
C05971=1012.588,7.020,-115.029,166.113,73.185,164.137
C05972=1012.588,7.250,-115.048,166.110,73.175,164.133
C05973=1012.587,7.478,-115.067,166.110,73.166,164.130
C05974=1012.587,7.704,-115.087,166.107,73.157,164.126
C05975=1012.587,7.929,-115.105,166.105,73.147,164.122
C05976=1012.587,8.153,-115.124,166.104,73.137,164.119
C05977=1012.587,8.377,-115.143,166.102,73.127,164.115
C05978=1012.587,8.601,-115.162,166.100,73.117,164.111
C05979=1012.587,8.823,-115.180,166.099,73.107,164.108
C05980=1012.586,9.045,-115.199,166.098,73.097,164.104
C05981=1012.586,9.268,-115.217,166.096,73.086,164.100
C05982=1012.587,9.491,-115.236,166.093,73.076,164.096
C05983=1012.587,9.713,-115.255,166.092,73.064,164.092
C05984=1012.586,9.937,-115.274,166.090,73.053,164.088
C05985=1012.586,10.160,-115.293,166.087,73.042,164.083
C05986=1012.586,10.384,-115.312,166.086,73.031,164.079
C05987=1012.586,10.609,-115.330,166.084,73.020,164.075
C05988=1012.586,10.834,-115.349,166.081,73.007,164.070
C05989=1012.586,11.055,-115.367,166.080,72.996,164.066
C05990=1012.586,11.273,-115.386,166.076,72.984,164.061
C05991=1012.586,11.489,-115.404,166.075,72.972,164.057
C05992=1012.586,11.705,-115.422,166.072,72.960,164.052
C05993=1012.586,11.924,-115.441,166.071,72.948,164.048
C05994=1012.585,12.148,-115.459,166.070,72.935,164.044
C05995=1012.586,12.375,-115.478,166.065,72.922,164.038
C05996=1012.585,12.604,-115.498,166.064,72.909,164.033
C05997=1012.585,12.832,-115.517,166.061,72.895,164.028
C05998=1012.585,13.061,-115.536,166.058,72.881,164.022
C05999=1012.585,13.290,-115.555,166.056,72.867,164.018
C06000=1012.585,13.517,-115.575,166.054,72.853,164.012
C06001=1012.586,13.745,-115.594,166.052,72.839,164.007
C06002=1012.584,13.972,-115.613,166.048,72.824,164.001
C06003=1012.585,14.199,-115.632,166.046,72.810,163.996
C06004=1012.584,14.426,-115.651,166.044,72.796,163.991
C06005=1012.584,14.652,-115.670,166.041,72.781,163.985
C06006=1012.585,14.878,-115.689,166.038,72.765,163.980
C06007=1012.584,15.104,-115.708,166.035,72.750,163.974
C06008=1012.584,15.330,-115.727,166.032,72.735,163.968
C06009=1012.584,15.557,-115.746,166.029,72.720,163.962
C06010=1012.584,15.783,-115.765,166.027,72.704,163.957
C06011=1012.584,16.011,-115.784,166.024,72.688,163.950
C06012=1012.584,16.237,-115.803,166.021,72.673,163.945
C06013=1012.584,16.465,-115.822,166.018,72.656,163.938
C06014=1012.584,16.692,-115.841,166.016,72.639,163.933
C06015=1012.584,16.921,-115.860,166.013,72.623,163.926
C06016=1012.584,17.150,-115.880,166.010,72.606,163.920
C06017=1012.584,17.380,-115.899,166.006,72.588,163.913
C06018=1012.584,17.611,-115.918,166.004,72.571,163.908
C06019=1012.584,17.842,-115.938,166.001,72.553,163.901
C06020=1012.584,18.074,-115.958,165.997,72.535,163.894
C06021=1012.584,18.306,-115.978,165.994,72.517,163.888
C06022=1012.584,18.539,-115.996,165.991,72.500,163.881
C06023=1012.584,18.773,-116.016,165.989,72.481,163.875
C06024=1012.583,19.006,-116.036,165.984,72.463,163.867
C06025=1012.583,19.268,-116.058,165.981,72.441,163.860
C06026=1012.584,19.573,-116.084,165.977,72.417,163.851
C06027=1012.584,19.969,-116.117,165.971,72.384,163.839
C06028=1012.584,20.269,-116.142,165.968,72.358,163.830
C06029=1012.584,20.588,-116.169,165.963,72.331,163.820
C06030=1012.584,20.908,-116.195,165.958,72.304,163.810
C06031=1012.584,21.217,-116.222,165.952,72.277,163.800
C06032=1012.584,21.506,-116.246,165.949,72.251,163.791
C06033=1012.583,21.766,-116.267,165.945,72.228,163.783
C06034=1012.583,22.177,-116.302,165.939,72.191,163.770
C06035=1012.583,22.590,-116.337,165.933,72.153,163.756
C06036=1012.583,22.935,-116.366,165.928,72.121,163.745
C06037=1012.584,23.226,-116.391,165.923,72.094,163.735
C06038=1012.584,23.527,-116.415,165.919,72.065,163.725
C06039=1012.583,23.891,-116.447,165.914,72.031,163.713
C06040=1012.583,24.100,-116.464,165.910,72.010,163.706
C06041=1012.584,24.323,-116.483,165.907,71.989,163.698
C06042=1012.584,24.555,-116.502,165.902,71.966,163.689
C06043=1012.584,24.791,-116.521,165.899,71.943,163.681
C06044=1012.583,25.027,-116.541,165.896,71.919,163.674
C06045=1012.583,25.262,-116.562,165.893,71.896,163.666
C06046=1012.583,25.498,-116.581,165.888,71.872,163.657
C06047=1012.584,25.734,-116.601,165.884,71.847,163.648
C06048=1012.584,25.972,-116.621,165.881,71.824,163.640
C06049=1012.584,26.208,-116.641,165.876,71.798,163.631
C06050=1012.583,26.445,-116.662,165.873,71.774,163.623
C06051=1012.583,26.681,-116.681,165.869,71.749,163.614
C06052=1012.584,26.917,-116.701,165.866,71.725,163.606
C06053=1012.583,27.151,-116.720,165.862,71.699,163.597
C06054=1012.584,27.386,-116.741,165.859,71.674,163.589
C06055=1012.584,27.620,-116.759,165.854,71.649,163.580
C06056=1012.583,27.854,-116.779,165.851,71.623,163.571
C06057=1012.584,28.088,-116.799,165.849,71.598,163.563
C06058=1012.584,28.322,-116.819,165.844,71.572,163.554
C06059=1012.584,28.556,-116.838,165.840,71.546,163.545
C06060=1012.584,28.791,-116.858,165.836,71.520,163.536
C06061=1012.584,29.026,-116.877,165.833,71.493,163.527
C06062=1012.584,29.261,-116.897,165.830,71.467,163.519
C06063=1012.584,29.497,-116.917,165.825,71.440,163.510
C06064=1012.584,29.732,-116.937,165.822,71.413,163.501
C06065=1012.584,29.967,-116.956,165.819,71.386,163.492
C06066=1012.584,30.202,-116.976,165.814,71.358,163.482
C06067=1012.584,30.438,-116.996,165.811,71.330,163.473
C06068=1012.585,30.673,-117.016,165.808,71.303,163.465
C06069=1012.584,30.908,-117.035,165.803,71.275,163.455
C06070=1012.584,31.143,-117.055,165.799,71.247,163.446
C06071=1012.584,31.379,-117.075,165.796,71.219,163.437
C06072=1012.585,31.614,-117.095,165.792,71.191,163.427
C06073=1012.585,31.850,-117.115,165.789,71.162,163.418
C06074=1012.585,32.085,-117.134,165.784,71.133,163.408
C06075=1012.584,32.321,-117.155,165.781,71.104,163.399
C06076=1012.584,32.556,-117.175,165.777,71.075,163.390
C06077=1012.584,32.792,-117.194,165.773,71.046,163.380
C06078=1012.585,33.027,-117.214,165.770,71.016,163.371
C06079=1012.584,33.262,-117.234,165.766,70.987,163.361
C06080=1012.585,33.497,-117.254,165.763,70.957,163.352
C06081=1012.585,33.733,-117.273,165.759,70.928,163.342
C06082=1012.585,33.968,-117.293,165.755,70.897,163.332
C06083=1012.585,34.204,-117.313,165.752,70.867,163.323
C06084=1012.585,34.440,-117.332,165.748,70.837,163.313
C06085=1012.585,34.674,-117.352,165.744,70.806,163.303
C06086=1012.585,34.910,-117.372,165.742,70.775,163.294
C06087=1012.585,35.145,-117.392,165.738,70.744,163.284
C06088=1012.585,35.381,-117.411,165.734,70.712,163.274
C06089=1012.586,35.616,-117.432,165.730,70.682,163.264
C06090=1012.586,35.852,-117.451,165.727,70.650,163.254
C06091=1012.586,36.087,-117.471,165.723,70.618,163.244
C06092=1012.585,36.322,-117.490,165.719,70.586,163.234
C06093=1012.586,36.557,-117.511,165.716,70.554,163.224
C06094=1012.586,36.793,-117.530,165.713,70.522,163.215
C06095=1012.586,37.028,-117.550,165.710,70.490,163.205
C06096=1012.586,37.264,-117.570,165.706,70.457,163.195
C06097=1012.587,37.499,-117.590,165.703,70.425,163.185
C06098=1012.586,37.837,-117.618,165.697,70.377,163.170
C06099=1012.587,38.205,-117.649,165.693,70.325,163.155
C06100=1012.587,38.441,-117.668,165.690,70.292,163.145
C06101=1012.587,38.676,-117.688,165.685,70.258,163.134
C06102=1012.587,38.912,-117.708,165.683,70.225,163.125
C06103=1012.587,39.147,-117.728,165.679,70.191,163.114
C06104=1012.587,39.383,-117.748,165.676,70.156,163.104
C06105=1012.588,39.618,-117.768,165.672,70.122,163.093
C06106=1012.588,39.854,-117.787,165.669,70.088,163.083
C06107=1012.588,40.090,-117.807,165.666,70.054,163.073
C06108=1012.588,40.325,-117.827,165.663,70.019,163.063
C06109=1012.588,40.561,-117.846,165.659,69.984,163.052
C06110=1012.589,40.796,-117.867,165.658,69.949,163.043
C06111=1012.589,41.031,-117.886,165.654,69.914,163.032
C06112=1012.589,41.267,-117.906,165.651,69.878,163.022
C06113=1012.589,41.502,-117.925,165.647,69.843,163.011
C06114=1012.589,41.737,-117.945,165.644,69.806,163.000
C06115=1012.589,41.973,-117.965,165.641,69.771,162.990
C06116=1012.589,42.208,-117.985,165.639,69.735,162.980
C06117=1012.589,42.444,-118.005,165.635,69.699,162.969
C06118=1012.589,42.679,-118.024,165.632,69.662,162.959
C06119=1012.590,42.915,-118.045,165.630,69.625,162.948
C06120=1012.590,43.150,-118.064,165.626,69.589,162.938
C06121=1012.590,43.386,-118.083,165.624,69.552,162.928
C06122=1012.590,43.621,-118.104,165.620,69.515,162.916
C06123=1012.590,43.857,-118.123,165.618,69.478,162.906
C06124=1012.591,44.092,-118.143,165.615,69.440,162.895
C06125=1012.591,44.328,-118.163,165.612,69.402,162.885
C06126=1012.591,44.564,-118.182,165.609,69.365,162.874
C06127=1012.591,44.799,-118.203,165.606,69.327,162.863
C06128=1012.591,45.035,-118.222,165.605,69.289,162.853
C06129=1012.592,45.270,-118.242,165.601,69.250,162.842
C06130=1012.592,45.506,-118.262,165.599,69.212,162.832
C06131=1012.593,45.742,-118.282,165.597,69.173,162.821
C06132=1012.593,45.977,-118.302,165.594,69.134,162.810
C06133=1012.593,46.213,-118.321,165.592,69.095,162.800
C06134=1012.593,46.448,-118.341,165.589,69.056,162.789
C06135=1012.593,46.684,-118.361,165.587,69.018,162.778
C06136=1012.593,46.920,-118.380,165.583,68.978,162.767
C06137=1012.593,47.155,-118.401,165.582,68.938,162.757
C06138=1012.593,47.391,-118.420,165.579,68.899,162.746
C06139=1012.594,47.626,-118.440,165.577,68.859,162.735
C06140=1012.594,47.862,-118.460,165.575,68.818,162.725
C06141=1012.594,48.098,-118.479,165.571,68.778,162.713
C06142=1012.594,48.333,-118.499,165.569,68.738,162.702
C06143=1012.595,48.569,-118.519,165.568,68.698,162.692
C06144=1012.595,48.805,-118.539,165.566,68.656,162.681
C06145=1012.595,49.040,-118.559,165.563,68.616,162.670
C06146=1012.595,49.276,-118.578,165.561,68.575,162.659
C06147=1012.596,49.511,-118.599,165.559,68.533,162.648
C06148=1012.596,49.747,-118.618,165.558,68.492,162.638
C06149=1012.596,49.983,-118.638,165.555,68.450,162.626
C06150=1012.597,50.219,-118.658,165.552,68.408,162.615
C06151=1012.597,50.454,-118.678,165.551,68.367,162.605
C06152=1012.597,50.690,-118.697,165.549,68.325,162.593
C06153=1012.597,50.925,-118.717,165.548,68.282,162.583
C06154=1012.597,51.161,-118.737,165.546,68.240,162.572
C06155=1012.597,51.397,-118.756,165.543,68.197,162.560
C06156=1012.598,51.633,-118.777,165.543,68.155,162.550
C06157=1012.598,51.869,-118.796,165.541,68.112,162.539
C06158=1012.599,52.104,-118.817,165.538,68.069,162.527
C06159=1012.599,52.340,-118.836,165.537,68.026,162.516
C06160=1012.599,52.575,-118.856,165.535,67.982,162.506
C06161=1012.600,52.811,-118.876,165.534,67.939,162.495
C06162=1012.600,53.047,-118.896,165.532,67.895,162.483
C06163=1012.600,53.283,-118.915,165.532,67.851,162.473
C06164=1012.600,53.518,-118.935,165.530,67.807,162.462
C06165=1012.600,53.754,-118.955,165.529,67.763,162.451
C06166=1012.601,53.990,-118.975,165.527,67.719,162.439
C06167=1012.601,54.226,-118.995,165.526,67.674,162.429
C06168=1012.601,54.461,-119.014,165.524,67.629,162.417
C06169=1012.601,54.697,-119.034,165.524,67.585,162.406
C06170=1012.602,54.933,-119.054,165.522,67.540,162.395
C06171=1012.603,55.169,-119.074,165.521,67.494,162.384
C06172=1012.603,55.405,-119.093,165.519,67.449,162.373
C06173=1012.603,55.640,-119.113,165.519,67.404,162.362
C06174=1012.604,55.876,-119.133,165.518,67.359,162.351
C06175=1012.604,56.112,-119.153,165.517,67.312,162.340
C06176=1012.604,56.347,-119.173,165.516,67.266,162.328
C06177=1012.604,56.583,-119.193,165.516,67.220,162.318
C06178=1012.605,56.819,-119.212,165.514,67.174,162.306
C06179=1012.605,57.055,-119.233,165.514,67.128,162.295
C06180=1012.605,57.290,-119.252,165.513,67.081,162.284
C06181=1012.606,57.527,-119.272,165.513,67.034,162.273
C06182=1012.606,57.762,-119.292,165.511,66.987,162.261
C06183=1012.606,57.998,-119.312,165.511,66.940,162.250
C06184=1012.606,58.234,-119.331,165.510,66.893,162.239
C06185=1012.607,58.470,-119.352,165.510,66.845,162.228
C06186=1012.607,58.705,-119.371,165.510,66.798,162.217
C06187=1012.608,58.940,-119.391,165.509,66.751,162.206
C06188=1012.608,59.177,-119.411,165.508,66.703,162.194
C06189=1012.608,59.413,-119.431,165.509,66.654,162.183
C06190=1012.609,59.648,-119.450,165.508,66.606,162.172
C06191=1012.610,59.884,-119.470,165.508,66.558,162.161
C06192=1012.610,60.120,-119.490,165.508,66.510,162.150
C06193=1012.610,60.355,-119.510,165.508,66.461,162.139
C06194=1012.610,60.591,-119.529,165.508,66.412,162.128
C06195=1012.611,60.827,-119.549,165.507,66.363,162.116
C06196=1012.612,61.063,-119.569,165.509,66.314,162.105
C06197=1012.612,61.298,-119.589,165.509,66.265,162.094
C06198=1012.612,61.535,-119.609,165.508,66.215,162.082
C06199=1012.613,61.770,-119.629,165.509,66.166,162.071
C06200=1012.613,62.006,-119.648,165.508,66.116,162.060
C06201=1012.614,62.242,-119.669,165.510,66.066,162.049
C06202=1012.614,62.518,-119.691,165.510,66.008,162.036
C06203=1012.615,62.805,-119.716,165.509,65.946,162.022
C06204=1012.615,63.081,-119.739,165.510,65.887,162.009
C06205=1012.616,63.377,-119.763,165.511,65.823,161.995
C06206=1012.617,63.660,-119.788,165.512,65.762,161.981
C06207=1012.617,63.911,-119.809,165.513,65.709,161.970
C06208=1012.618,64.148,-119.828,165.514,65.657,161.958
C06209=1012.617,64.402,-119.850,165.515,65.602,161.946
C06210=1012.618,64.669,-119.872,165.516,65.543,161.933
C06211=1012.618,64.939,-119.896,165.517,65.484,161.921
C06212=1012.619,65.204,-119.917,165.518,65.426,161.908
C06213=1012.620,65.465,-119.939,165.518,65.368,161.895
C06214=1012.621,65.719,-119.960,165.520,65.312,161.883
C06215=1012.621,65.961,-119.981,165.521,65.258,161.872
C06216=1012.622,66.193,-120.000,165.522,65.207,161.860
C06217=1012.622,66.586,-120.033,165.524,65.119,161.842
C06218=1012.623,66.800,-120.051,165.525,65.070,161.831
C06219=1012.623,67.035,-120.071,165.526,65.018,161.820
C06220=1012.624,67.272,-120.092,165.528,64.964,161.809
C06221=1012.624,67.510,-120.111,165.529,64.910,161.797
C06222=1012.625,67.826,-120.138,165.531,64.838,161.782
C06223=1012.626,68.228,-120.171,165.534,64.747,161.763
C06224=1012.627,68.473,-120.192,165.536,64.691,161.751
C06225=1012.627,68.722,-120.213,165.538,64.634,161.739
C06226=1012.627,68.971,-120.234,165.539,64.576,161.727
C06227=1012.628,69.220,-120.255,165.542,64.518,161.716
C06228=1012.628,69.465,-120.276,165.544,64.461,161.704
C06229=1012.629,69.709,-120.296,165.546,64.406,161.692
C06230=1012.630,69.951,-120.316,165.548,64.349,161.681
C06231=1012.630,70.191,-120.337,165.550,64.292,161.669
C06232=1012.630,70.432,-120.357,165.553,64.236,161.658
C06233=1012.632,70.673,-120.377,165.555,64.180,161.646
C06234=1012.632,70.914,-120.397,165.556,64.122,161.634
C06235=1012.633,71.156,-120.419,165.559,64.065,161.623
C06236=1012.633,71.397,-120.439,165.562,64.009,161.611
C06237=1012.634,71.638,-120.458,165.564,63.951,161.600
C06238=1012.635,71.879,-120.479,165.567,63.894,161.588
C06239=1012.635,72.121,-120.499,165.569,63.836,161.576
C06240=1012.636,72.362,-120.520,165.572,63.778,161.565
C06241=1012.636,72.605,-120.539,165.575,63.719,161.553
C06242=1012.637,72.848,-120.561,165.578,63.661,161.541
C06243=1012.638,73.091,-120.581,165.581,63.602,161.530
C06244=1012.639,73.335,-120.602,165.584,63.543,161.518
C06245=1012.639,73.580,-120.622,165.586,63.484,161.506
C06246=1012.640,73.826,-120.643,165.590,63.424,161.495
C06247=1012.641,74.073,-120.663,165.593,63.364,161.483
C06248=1012.641,74.323,-120.685,165.597,63.302,161.471
C06249=1012.641,74.591,-120.707,165.599,63.236,161.457
C06250=1012.643,74.864,-120.730,165.604,63.169,161.444
C06251=1012.644,75.122,-120.752,165.608,63.105,161.432
C06252=1012.644,75.371,-120.773,165.610,63.043,161.420
C06253=1012.644,75.619,-120.793,165.614,62.982,161.408
C06254=1012.645,75.864,-120.814,165.619,62.921,161.396
C06255=1012.646,76.109,-120.835,165.622,62.860,161.385
C06256=1012.647,76.349,-120.855,165.626,62.799,161.373
C06257=1012.648,76.588,-120.876,165.629,62.740,161.361
C06258=1012.648,76.824,-120.895,165.633,62.681,161.350
C06259=1012.649,77.056,-120.914,165.637,62.622,161.339
C06260=1012.650,77.287,-120.934,165.641,62.563,161.328
C06261=1012.651,77.515,-120.953,165.645,62.505,161.317
C06262=1012.651,77.743,-120.972,165.649,62.448,161.306
C06263=1012.652,77.970,-120.992,165.653,62.390,161.295
C06264=1012.653,78.197,-121.011,165.657,62.332,161.284
C06265=1012.653,78.427,-121.030,165.661,62.273,161.273
C06266=1012.654,78.657,-121.049,165.664,62.214,161.262
C06267=1012.654,78.889,-121.069,165.669,62.154,161.250
C06268=1012.656,79.124,-121.089,165.674,62.093,161.239
C06269=1012.657,79.362,-121.109,165.678,62.032,161.228
C06270=1012.657,79.601,-121.129,165.683,61.970,161.216
C06271=1012.657,79.843,-121.150,165.687,61.907,161.204
C06272=1012.659,80.087,-121.170,165.692,61.843,161.192
C06273=1012.659,80.334,-121.191,165.696,61.779,161.180
C06274=1012.661,80.577,-121.211,165.702,61.716,161.169
C06275=1012.661,80.807,-121.231,165.706,61.656,161.158
C06276=1012.661,81.023,-121.249,165.711,61.598,161.147
C06277=1012.663,81.241,-121.267,165.715,61.541,161.137
C06278=1012.664,81.469,-121.286,165.721,61.481,161.126
C06279=1012.664,81.712,-121.307,165.726,61.417,161.114
C06280=1012.664,81.959,-121.328,165.731,61.351,161.102
C06281=1012.666,82.206,-121.349,165.737,61.286,161.090
C06282=1012.667,82.453,-121.370,165.742,61.220,161.078
C06283=1012.668,82.699,-121.390,165.747,61.154,161.066
C06284=1012.669,82.946,-121.411,165.753,61.088,161.054
C06285=1012.670,83.191,-121.432,165.758,61.022,161.042
C06286=1012.670,83.436,-121.452,165.765,60.956,161.031
C06287=1012.671,83.681,-121.474,165.771,60.890,161.019
C06288=1012.672,83.926,-121.494,165.776,60.824,161.007
C06289=1012.673,84.170,-121.515,165.782,60.758,160.995
C06290=1012.674,84.413,-121.535,165.789,60.692,160.983
C06291=1012.675,84.656,-121.556,165.794,60.625,160.971
C06292=1012.675,84.900,-121.576,165.800,60.559,160.959
C06293=1012.676,85.142,-121.597,165.807,60.494,160.948
C06294=1012.678,85.384,-121.617,165.812,60.427,160.936
C06295=1012.678,85.624,-121.637,165.818,60.361,160.924
C06296=1012.680,85.865,-121.658,165.825,60.294,160.912
C06297=1012.681,86.105,-121.678,165.832,60.228,160.901
C06298=1012.681,86.345,-121.698,165.838,60.162,160.889
C06299=1012.682,86.585,-121.719,165.844,60.095,160.877
C06300=1012.683,86.824,-121.738,165.851,60.029,160.865
C06301=1012.684,87.063,-121.759,165.857,59.963,160.854
C06302=1012.685,87.300,-121.779,165.864,59.896,160.842
C06303=1012.686,87.536,-121.799,165.871,59.830,160.831
C06304=1012.687,87.771,-121.818,165.878,59.764,160.819
C06305=1012.687,88.001,-121.838,165.885,59.700,160.808
C06306=1012.689,88.228,-121.858,165.891,59.636,160.797
C06307=1012.689,88.453,-121.876,165.898,59.573,160.786
C06308=1012.691,88.677,-121.895,165.905,59.510,160.775
C06309=1012.692,89.058,-121.928,165.916,59.402,160.756
C06310=1012.693,89.218,-121.941,165.920,59.357,160.748
C06311=1012.781,44.749,-117.778,165.692,60.251,160.861
C06312=1012.782,44.367,-117.746,165.685,60.314,160.872
C06313=1012.780,44.131,-117.726,165.681,60.351,160.879
C06314=1012.780,43.896,-117.706,165.678,60.389,160.885
C06315=1012.779,43.660,-117.686,165.674,60.426,160.892
C06316=1012.779,43.425,-117.666,165.670,60.463,160.898
C06317=1012.779,43.189,-117.646,165.666,60.500,160.904
C06318=1012.778,42.954,-117.626,165.662,60.537,160.911
C06319=1012.778,42.718,-117.606,165.658,60.574,160.917
C06320=1012.777,42.483,-117.587,165.655,60.611,160.924
C06321=1012.777,42.247,-117.567,165.651,60.647,160.930
C06322=1012.777,42.012,-117.547,165.649,60.683,160.936
C06323=1012.776,41.776,-117.528,165.644,60.719,160.942
C06324=1012.776,41.540,-117.507,165.641,60.755,160.949
C06325=1012.775,41.305,-117.487,165.638,60.790,160.955
C06326=1012.775,41.069,-117.467,165.633,60.826,160.961
C06327=1012.774,40.834,-117.448,165.630,60.861,160.967
C06328=1012.774,40.599,-117.428,165.627,60.896,160.973
C06329=1012.774,40.363,-117.408,165.623,60.931,160.979
C06330=1012.774,40.128,-117.389,165.620,60.966,160.986
C06331=1012.773,39.892,-117.368,165.617,61.001,160.992
C06332=1012.772,39.657,-117.348,165.614,61.035,160.998
C06333=1012.772,39.421,-117.328,165.611,61.070,161.004
C06334=1012.771,39.186,-117.309,165.607,61.104,161.010
C06335=1012.771,38.950,-117.289,165.604,61.137,161.016
C06336=1012.771,38.715,-117.269,165.601,61.171,161.021
C06337=1012.771,38.479,-117.250,165.598,61.205,161.028
C06338=1012.770,38.244,-117.229,165.595,61.238,161.034
C06339=1012.770,38.009,-117.209,165.591,61.271,161.039
C06340=1012.770,37.773,-117.190,165.588,61.305,161.045
C06341=1012.769,37.538,-117.169,165.585,61.337,161.051
C06342=1012.768,37.302,-117.150,165.582,61.371,161.057
C06343=1012.768,37.067,-117.130,165.579,61.403,161.063
C06344=1012.768,36.831,-117.110,165.577,61.435,161.068
C06345=1012.767,36.596,-117.090,165.573,61.467,161.074
C06346=1012.767,36.361,-117.070,165.570,61.500,161.080
C06347=1012.767,36.125,-117.051,165.567,61.531,161.085
C06348=1012.767,35.890,-117.030,165.565,61.564,161.091
C06349=1012.766,35.654,-117.011,165.561,61.595,161.097
C06350=1012.766,35.419,-116.991,165.560,61.626,161.102
C06351=1012.765,35.184,-116.971,165.556,61.657,161.107
C06352=1012.765,34.948,-116.952,165.554,61.688,161.113
C06353=1012.765,34.713,-116.931,165.550,61.719,161.119
C06354=1012.765,34.477,-116.912,165.548,61.750,161.124
C06355=1012.764,34.242,-116.892,165.545,61.780,161.129
C06356=1012.764,34.006,-116.872,165.542,61.810,161.135
C06357=1012.764,33.771,-116.852,165.540,61.841,161.140
C06358=1012.763,33.536,-116.832,165.537,61.871,161.146
C06359=1012.763,33.300,-116.812,165.534,61.901,161.151
C06360=1012.762,33.065,-116.793,165.532,61.930,161.156
C06361=1012.762,32.829,-116.773,165.529,61.960,161.162
C06362=1012.762,32.594,-116.753,165.527,61.989,161.167
C06363=1012.762,32.359,-116.733,165.524,62.018,161.172
C06364=1012.761,32.123,-116.713,165.522,62.047,161.178
C06365=1012.761,31.888,-116.693,165.520,62.076,161.183
C06366=1012.761,31.652,-116.674,165.517,62.104,161.188
C06367=1012.761,31.417,-116.654,165.514,62.133,161.193
C06368=1012.760,31.182,-116.633,165.512,62.161,161.198
C06369=1012.760,30.946,-116.614,165.509,62.189,161.203
C06370=1012.761,30.712,-116.594,165.507,62.217,161.208
C06371=1012.760,30.476,-116.575,165.505,62.244,161.213
C06372=1012.759,30.241,-116.555,165.502,62.272,161.218
C06373=1012.759,30.005,-116.535,165.500,62.299,161.223
C06374=1012.759,29.770,-116.515,165.498,62.327,161.228
C06375=1012.759,29.535,-116.495,165.495,62.353,161.232
C06376=1012.759,29.299,-116.476,165.493,62.381,161.237
C06377=1012.758,29.064,-116.455,165.491,62.407,161.242
C06378=1012.758,28.829,-116.435,165.489,62.433,161.247
C06379=1012.757,28.595,-116.416,165.487,62.460,161.252
C06380=1012.758,28.360,-116.396,165.484,62.485,161.256
C06381=1012.757,28.126,-116.377,165.483,62.511,161.261
C06382=1012.757,27.892,-116.357,165.480,62.537,161.266
C06383=1012.756,27.658,-116.337,165.478,62.562,161.270
C06384=1012.757,27.424,-116.317,165.475,62.588,161.275
C06385=1012.756,27.190,-116.298,165.474,62.613,161.280
C06386=1012.756,26.955,-116.278,165.472,62.638,161.284
C06387=1012.756,26.719,-116.258,165.470,62.662,161.289
C06388=1012.755,26.483,-116.238,165.467,62.688,161.293
C06389=1012.756,26.246,-116.218,165.465,62.712,161.298
C06390=1012.755,26.009,-116.199,165.463,62.736,161.302
C06391=1012.755,25.771,-116.178,165.462,62.760,161.306
C06392=1012.756,25.535,-116.158,165.460,62.785,161.311
C06393=1012.755,25.300,-116.138,165.457,62.808,161.315
C06394=1012.755,25.065,-116.119,165.455,62.833,161.319
C06395=1012.755,24.828,-116.099,165.453,62.856,161.324
C06396=1012.754,24.593,-116.079,165.451,62.879,161.328
C06397=1012.755,24.360,-116.059,165.450,62.902,161.332
C06398=1012.754,24.138,-116.041,165.447,62.923,161.336
C06399=1012.754,23.929,-116.024,165.446,62.944,161.340
C06400=1012.753,23.565,-115.992,165.443,62.978,161.346
C06401=1012.753,23.264,-115.967,165.440,63.007,161.351
C06402=1012.753,22.972,-115.942,165.438,63.034,161.356
C06403=1012.753,22.627,-115.914,165.436,63.066,161.362
C06404=1012.753,22.214,-115.879,165.433,63.104,161.369
C06405=1012.753,21.803,-115.844,165.430,63.141,161.376
C06406=1012.753,21.544,-115.822,165.428,63.163,161.380
C06407=1012.752,21.255,-115.798,165.426,63.189,161.384
C06408=1012.751,20.946,-115.772,165.424,63.216,161.389
C06409=1012.752,20.626,-115.745,165.421,63.243,161.394
C06410=1012.752,20.307,-115.718,165.419,63.270,161.399
C06411=1012.751,20.007,-115.693,165.417,63.296,161.404
C06412=1012.751,19.611,-115.660,165.414,63.328,161.409
C06413=1012.751,19.306,-115.633,165.412,63.353,161.414
C06414=1012.751,19.043,-115.612,165.410,63.374,161.418
C06415=1012.751,18.810,-115.592,165.408,63.392,161.421
C06416=1012.751,18.576,-115.573,165.407,63.411,161.425
C06417=1012.750,18.343,-115.553,165.405,63.429,161.428
C06418=1012.751,18.111,-115.534,165.404,63.447,161.431
C06419=1012.750,17.879,-115.513,165.402,63.465,161.435
C06420=1012.750,17.649,-115.494,165.400,63.482,161.437
C06421=1012.750,17.417,-115.475,165.400,63.499,161.441
C06422=1012.751,17.188,-115.455,165.398,63.517,161.444
C06423=1012.750,16.959,-115.436,165.396,63.534,161.447
C06424=1012.750,16.730,-115.417,165.394,63.551,161.450
C06425=1012.749,16.502,-115.398,165.394,63.567,161.453
C06426=1012.749,16.275,-115.379,165.391,63.583,161.456
C06427=1012.750,16.048,-115.359,165.391,63.599,161.459
C06428=1012.749,15.820,-115.341,165.389,63.615,161.462
C06429=1012.749,15.594,-115.321,165.387,63.630,161.464
C06430=1012.750,15.368,-115.302,165.386,63.646,161.467
C06431=1012.750,15.142,-115.283,165.385,63.661,161.470
C06432=1012.749,14.916,-115.264,165.383,63.676,161.472
C06433=1012.749,14.690,-115.245,165.382,63.691,161.475
C06434=1012.750,14.463,-115.226,165.380,63.705,161.478
C06435=1012.750,14.236,-115.207,165.378,63.720,161.480
C06436=1012.750,14.009,-115.188,165.377,63.734,161.483
C06437=1012.749,13.782,-115.169,165.376,63.748,161.486
C06438=1012.749,13.555,-115.150,165.375,63.762,161.488
C06439=1012.750,13.326,-115.131,165.374,63.777,161.491
C06440=1012.749,13.098,-115.111,165.373,63.790,161.493
C06441=1012.749,12.869,-115.092,165.372,63.804,161.496
C06442=1012.749,12.640,-115.073,165.370,63.818,161.498
C06443=1012.749,12.412,-115.053,165.368,63.831,161.500
C06444=1012.749,12.185,-115.034,165.367,63.844,161.503
C06445=1012.749,11.961,-115.016,165.366,63.856,161.505
C06446=1012.749,11.742,-114.997,165.364,63.868,161.507
C06447=1012.749,11.525,-114.979,165.363,63.880,161.509
C06448=1012.749,11.310,-114.961,165.362,63.892,161.511
C06449=1012.749,11.092,-114.942,165.361,63.904,161.513
C06450=1012.749,10.871,-114.923,165.360,63.915,161.515
C06451=1012.749,10.646,-114.905,165.358,63.927,161.517
C06452=1012.749,10.421,-114.886,165.357,63.938,161.519
C06453=1012.749,10.197,-114.868,165.356,63.950,161.521
C06454=1012.749,9.973,-114.848,165.354,63.961,161.523
C06455=1012.750,9.750,-114.829,165.353,63.972,161.525
C06456=1012.749,9.527,-114.811,165.352,63.983,161.527
C06457=1012.750,9.304,-114.792,165.351,63.993,161.529
C06458=1012.749,9.082,-114.773,165.350,64.004,161.530
C06459=1012.749,8.860,-114.755,165.348,64.014,161.532
C06460=1012.749,8.637,-114.736,165.348,64.024,161.534
C06461=1012.749,8.415,-114.717,165.347,64.034,161.536
C06462=1012.749,8.191,-114.699,165.345,64.044,161.537
C06463=1012.749,7.966,-114.679,165.343,64.053,161.538
C06464=1012.750,7.741,-114.660,165.342,64.063,161.540
C06465=1012.750,7.514,-114.642,165.341,64.072,161.542
C06466=1012.750,7.287,-114.623,165.339,64.081,161.543
C06467=1012.749,7.057,-114.603,165.339,64.089,161.545
C06468=1012.749,6.827,-114.584,165.338,64.099,161.546
C06469=1012.750,6.593,-114.564,165.336,64.108,161.548
C06470=1012.750,6.360,-114.545,165.335,64.116,161.549
C06471=1012.750,6.126,-114.524,165.335,64.125,161.551
C06472=1012.749,5.892,-114.505,165.332,64.133,161.552
C06473=1012.750,5.658,-114.486,165.331,64.141,161.553
C06474=1012.750,5.426,-114.465,165.330,64.149,161.554
C06475=1012.750,5.194,-114.446,165.328,64.157,161.555
C06476=1012.750,4.963,-114.427,165.328,64.164,161.557
C06477=1012.750,4.731,-114.408,165.326,64.171,161.558
C06478=1012.750,4.499,-114.388,165.326,64.178,161.559
C06479=1012.751,4.266,-114.368,165.324,64.185,161.560
C06480=1012.750,4.037,-114.349,165.323,64.192,161.561
C06481=1012.751,3.819,-114.331,165.323,64.198,161.562
C06482=1012.751,3.610,-114.313,165.321,64.204,161.563
C06483=1012.751,3.218,-114.280,165.319,64.214,161.564
C06484=1012.751,2.834,-114.247,165.316,64.224,161.565
C06485=1012.750,2.425,-114.213,165.315,64.233,161.567
C06486=1012.751,2.205,-114.195,165.314,64.238,161.568
C06487=1012.751,1.976,-114.175,165.313,64.243,161.568
C06488=1012.751,1.741,-114.155,165.311,64.248,161.568
C06489=1012.752,1.504,-114.136,165.310,64.253,161.569
C06490=1012.751,1.268,-114.116,165.309,64.257,161.569
C06491=1012.752,1.031,-114.096,165.309,64.262,161.570
C06492=1012.752,0.797,-114.076,165.308,64.266,161.571
C06493=1012.752,0.562,-114.056,165.305,64.269,161.571
C06494=1012.752,0.327,-114.037,165.305,64.273,161.571
C06495=1012.752,0.092,-114.017,165.304,64.277,161.572
C06496=1012.753,-0.146,-113.997,165.302,64.280,161.572
C06497=1012.753,-0.383,-113.977,165.301,64.283,161.572
C06498=1012.753,-0.621,-113.957,165.300,64.285,161.572
C06499=1012.753,-0.861,-113.937,165.298,64.289,161.572
C06500=1012.753,-1.101,-113.916,165.298,64.291,161.573
C06501=1012.753,-1.342,-113.896,165.297,64.293,161.572
C06502=1012.753,-1.583,-113.876,165.296,64.295,161.573
C06503=1012.754,-1.825,-113.856,165.295,64.297,161.573
C06504=1012.754,-2.068,-113.835,165.293,64.299,161.573
C06505=1012.754,-2.311,-113.815,165.292,64.301,161.572
C06506=1012.754,-2.556,-113.794,165.291,64.301,161.572
C06507=1012.754,-2.800,-113.773,165.289,64.303,161.572
C06508=1012.755,-3.046,-113.753,165.288,64.304,161.572
C06509=1012.755,-3.288,-113.732,165.287,64.304,161.571
C06510=1012.755,-3.525,-113.713,165.286,64.305,161.571
C06511=1012.755,-3.756,-113.694,165.285,64.305,161.571
C06512=1012.755,-3.982,-113.674,165.284,64.304,161.570
C06513=1012.756,-4.207,-113.655,165.283,64.305,161.570
C06514=1012.755,-4.436,-113.636,165.282,64.304,161.569
C06515=1012.756,-4.672,-113.616,165.280,64.304,161.569
C06516=1012.756,-4.916,-113.596,165.279,64.303,161.568
C06517=1012.756,-5.168,-113.574,165.279,64.301,161.567
C06518=1012.756,-5.425,-113.553,165.278,64.300,161.567
C06519=1012.757,-5.683,-113.532,165.276,64.299,161.566
C06520=1012.757,-5.941,-113.509,165.275,64.297,161.565
C06521=1012.758,-6.199,-113.488,165.273,64.295,161.564
C06522=1012.757,-6.457,-113.466,165.272,64.293,161.563
C06523=1012.758,-6.714,-113.445,165.270,64.290,161.562
C06524=1012.757,-6.970,-113.423,165.270,64.287,161.561
C06525=1012.758,-7.226,-113.401,165.269,64.284,161.560
C06526=1012.758,-7.480,-113.379,165.267,64.281,161.559
C06527=1012.759,-7.733,-113.358,165.266,64.277,161.557
C06528=1012.759,-7.986,-113.338,165.265,64.273,161.556
C06529=1012.759,-8.238,-113.316,165.264,64.270,161.555
C06530=1012.759,-8.490,-113.295,165.262,64.265,161.553
C06531=1012.760,-8.740,-113.274,165.261,64.261,161.552
C06532=1012.760,-8.992,-113.253,165.261,64.256,161.551
C06533=1012.760,-9.243,-113.232,165.259,64.251,161.549
C06534=1012.760,-9.495,-113.211,165.258,64.246,161.548
C06535=1012.760,-9.746,-113.190,165.257,64.241,161.546
C06536=1012.761,-9.996,-113.169,165.256,64.235,161.545
C06537=1012.762,-10.246,-113.148,165.254,64.229,161.543
C06538=1012.762,-10.497,-113.126,165.253,64.223,161.541
C06539=1012.762,-10.746,-113.106,165.252,64.217,161.539
C06540=1012.762,-10.995,-113.084,165.250,64.210,161.537
C06541=1012.763,-11.244,-113.063,165.250,64.203,161.535
C06542=1012.763,-11.492,-113.043,165.249,64.197,161.534
C06543=1012.763,-11.739,-113.022,165.247,64.190,161.532
C06544=1012.764,-11.986,-113.001,165.246,64.182,161.529
C06545=1012.764,-12.233,-112.981,165.245,64.174,161.528
C06546=1012.765,-12.478,-112.959,165.245,64.166,161.526
C06547=1012.765,-12.723,-112.939,165.243,64.159,161.524
C06548=1012.765,-12.965,-112.918,165.242,64.150,161.521
C06549=1012.765,-13.202,-112.899,165.241,64.143,161.519
C06550=1012.765,-13.435,-112.879,165.240,64.134,161.517
C06551=1012.766,-13.664,-112.859,165.240,64.126,161.515
C06552=1012.766,-13.890,-112.841,165.238,64.117,161.513
C06553=1012.767,-14.114,-112.822,165.237,64.109,161.510
C06554=1012.766,-14.337,-112.803,165.236,64.100,161.508
C06555=1012.767,-14.560,-112.785,165.234,64.092,161.506
C06556=1012.768,-14.785,-112.765,165.234,64.082,161.504
C06557=1012.768,-15.011,-112.746,165.232,64.073,161.501
C06558=1012.768,-15.242,-112.727,165.231,64.063,161.498
C06559=1012.769,-15.474,-112.707,165.231,64.053,161.496
C06560=1012.769,-15.710,-112.688,165.229,64.042,161.493
C06561=1012.770,-15.946,-112.668,165.229,64.032,161.491
C06562=1012.770,-16.182,-112.648,165.227,64.021,161.488
C06563=1012.770,-16.416,-112.629,165.226,64.010,161.485
C06564=1012.770,-16.654,-112.609,165.226,63.999,161.483
C06565=1012.771,-16.892,-112.589,165.224,63.987,161.480
C06566=1012.772,-17.126,-112.569,165.223,63.976,161.477
C06567=1012.772,-17.357,-112.550,165.222,63.964,161.474
C06568=1012.772,-17.588,-112.530,165.222,63.952,161.472
C06569=1012.773,-17.835,-112.509,165.221,63.939,161.468
C06570=1012.773,-18.119,-112.485,165.219,63.924,161.464
C06571=1012.773,-18.437,-112.458,165.218,63.906,161.460
C06572=1012.774,-18.770,-112.430,165.216,63.888,161.456
C06573=1012.775,-19.095,-112.403,165.215,63.869,161.451
C06574=1012.775,-19.394,-112.378,165.214,63.852,161.447
C06575=1012.775,-19.655,-112.356,165.213,63.836,161.444
C06576=1012.776,-20.005,-112.327,165.211,63.815,161.438
C06577=1012.777,-20.283,-112.304,165.211,63.798,161.435
C06578=1012.777,-20.517,-112.284,165.209,63.783,161.431
C06579=1012.777,-20.752,-112.264,165.208,63.768,161.427
C06580=1012.778,-20.986,-112.245,165.208,63.753,161.424
C06581=1012.778,-21.220,-112.225,165.206,63.738,161.420
C06582=1012.779,-21.454,-112.205,165.205,63.722,161.416
C06583=1012.779,-21.688,-112.186,165.204,63.706,161.413
C06584=1012.780,-21.923,-112.166,165.204,63.691,161.409
C06585=1012.780,-22.156,-112.146,165.202,63.674,161.405
C06586=1012.781,-22.391,-112.126,165.202,63.657,161.402
C06587=1012.781,-22.625,-112.107,165.201,63.641,161.398
C06588=1012.782,-22.859,-112.087,165.200,63.624,161.394
C06589=1012.782,-23.094,-112.067,165.200,63.607,161.390
C06590=1012.783,-23.327,-112.048,165.199,63.589,161.386
C06591=1012.783,-23.562,-112.028,165.198,63.572,161.382
C06592=1012.784,-23.796,-112.009,165.197,63.554,161.378
C06593=1012.784,-24.030,-111.989,165.195,63.536,161.374
C06594=1012.784,-24.264,-111.969,165.195,63.518,161.370
C06595=1012.785,-24.498,-111.949,165.194,63.500,161.365
C06596=1012.785,-24.733,-111.930,165.193,63.481,161.361
C06597=1012.786,-24.966,-111.910,165.192,63.462,161.357
C06598=1012.786,-25.201,-111.890,165.191,63.443,161.353
C06599=1012.787,-25.435,-111.870,165.192,63.424,161.349
C06600=1012.788,-25.669,-111.851,165.190,63.404,161.344
C06601=1012.789,-25.904,-111.831,165.189,63.385,161.340
C06602=1012.789,-26.137,-111.811,165.189,63.365,161.335
C06603=1012.790,-26.372,-111.791,165.188,63.344,161.331
C06604=1012.790,-26.606,-111.771,165.187,63.324,161.326
C06605=1012.791,-26.840,-111.752,165.186,63.303,161.322
C06606=1012.791,-27.075,-111.732,165.186,63.283,161.317
C06607=1012.792,-27.308,-111.713,165.186,63.261,161.313
C06608=1012.792,-27.543,-111.693,165.184,63.240,161.307
C06609=1012.792,-27.777,-111.673,165.184,63.218,161.303
C06610=1012.793,-28.011,-111.654,165.183,63.196,161.298
C06611=1012.793,-28.245,-111.634,165.182,63.175,161.293
C06612=1012.794,-28.481,-111.615,165.182,63.153,161.289
C06613=1012.795,-28.715,-111.595,165.181,63.130,161.283
C06614=1012.796,-28.949,-111.575,165.180,63.108,161.279
C06615=1012.797,-29.183,-111.555,165.180,63.084,161.274
C06616=1012.797,-29.417,-111.535,165.179,63.061,161.269
C06617=1012.797,-29.652,-111.516,165.178,63.038,161.263
C06618=1012.798,-29.885,-111.496,165.178,63.015,161.258
C06619=1012.798,-30.120,-111.476,165.177,62.991,161.253
C06620=1012.799,-30.354,-111.457,165.177,62.967,161.248
C06621=1012.800,-30.589,-111.437,165.176,62.943,161.243
C06622=1012.800,-30.823,-111.417,165.176,62.918,161.238
C06623=1012.801,-31.057,-111.398,165.175,62.894,161.232
C06624=1012.802,-31.292,-111.378,165.174,62.869,161.227
C06625=1012.802,-31.525,-111.359,165.174,62.843,161.221
C06626=1012.803,-31.760,-111.339,165.174,62.819,161.216
C06627=1012.804,-31.995,-111.318,165.174,62.792,161.211
C06628=1012.804,-32.228,-111.299,165.173,62.767,161.205
C06629=1012.805,-32.463,-111.280,165.173,62.740,161.200
C06630=1012.806,-32.697,-111.260,165.172,62.715,161.194
C06631=1012.806,-32.932,-111.240,165.172,62.688,161.189
C06632=1012.807,-33.166,-111.220,165.171,62.661,161.183
C06633=1012.808,-33.400,-111.201,165.171,62.635,161.177
C06634=1012.808,-33.635,-111.181,165.171,62.607,161.172
C06635=1012.809,-33.869,-111.162,165.170,62.579,161.166
C06636=1012.809,-34.103,-111.142,165.170,62.552,161.160
C06637=1012.810,-34.338,-111.122,165.169,62.524,161.154
C06638=1012.811,-34.572,-111.102,165.169,62.496,161.148
C06639=1012.812,-34.806,-111.082,165.169,62.468,161.143
C06640=1012.812,-35.040,-111.063,165.169,62.440,161.137
C06641=1012.813,-35.275,-111.043,165.170,62.411,161.131
C06642=1012.814,-35.509,-111.024,165.168,62.382,161.125
C06643=1012.815,-35.744,-111.004,165.169,62.353,161.119
C06644=1012.816,-35.977,-110.984,165.168,62.323,161.113
C06645=1012.816,-36.212,-110.965,165.168,62.294,161.107
C06646=1012.817,-36.446,-110.945,165.167,62.263,161.100
C06647=1012.818,-36.680,-110.925,165.167,62.234,161.094
C06648=1012.819,-36.915,-110.906,165.168,62.203,161.088
C06649=1012.819,-37.149,-110.886,165.167,62.172,161.082
C06650=1012.820,-37.383,-110.867,165.168,62.142,161.075
C06651=1012.821,-37.618,-110.846,165.167,62.111,161.069
C06652=1012.822,-37.851,-110.827,165.167,62.080,161.063
C06653=1012.822,-38.086,-110.807,165.167,62.048,161.056
C06654=1012.823,-38.320,-110.787,165.168,62.016,161.050
C06655=1012.824,-38.555,-110.768,165.168,61.984,161.043
C06656=1012.825,-38.789,-110.748,165.167,61.952,161.037
C06657=1012.825,-39.023,-110.728,165.168,61.919,161.030
C06658=1012.826,-39.257,-110.709,165.168,61.886,161.024
C06659=1012.827,-39.492,-110.689,165.169,61.854,161.017
C06660=1012.828,-39.725,-110.669,165.169,61.821,161.011
C06661=1012.829,-39.959,-110.650,165.169,61.787,161.004
C06662=1012.829,-40.194,-110.631,165.169,61.754,160.997
C06663=1012.831,-40.428,-110.610,165.170,61.720,160.990
C06664=1012.831,-40.663,-110.591,165.169,61.686,160.983
C06665=1012.832,-40.897,-110.571,165.170,61.652,160.977
C06666=1012.833,-41.130,-110.552,165.170,61.617,160.970
C06667=1012.834,-41.365,-110.531,165.170,61.582,160.963
C06668=1012.834,-41.599,-110.512,165.171,61.548,160.956
C06669=1012.835,-41.833,-110.492,165.171,61.512,160.949
C06670=1012.836,-42.068,-110.473,165.171,61.476,160.942
C06671=1012.837,-42.302,-110.453,165.171,61.441,160.935
C06672=1012.838,-42.535,-110.434,165.172,61.405,160.928
C06673=1012.839,-42.770,-110.414,165.172,61.369,160.921
C06674=1012.839,-43.004,-110.394,165.174,61.333,160.914
C06675=1012.841,-43.238,-110.374,165.174,61.296,160.907
C06676=1012.842,-43.471,-110.355,165.174,61.259,160.899
C06677=1012.842,-43.706,-110.335,165.175,61.222,160.892
C06678=1012.843,-43.940,-110.316,165.176,61.184,160.885
C06679=1012.844,-44.174,-110.296,165.176,61.147,160.877
C06680=1012.845,-44.389,-110.278,165.177,61.112,160.871
C06681=1012.498,-134.033,-105.667,-74.106,87.342,-74.071
C06682=1012.498,-133.687,-105.696,-71.135,87.216,-71.096
C06683=1012.499,-133.340,-105.726,-68.436,87.084,-68.391
C06684=1012.498,-133.109,-105.745,-66.768,86.992,-66.720
C06685=1012.499,-132.878,-105.764,-65.214,86.899,-65.162
C06686=1012.498,-132.647,-105.784,-63.739,86.803,-63.684
C06687=1012.499,-132.416,-105.803,-62.364,86.705,-62.306
C06688=1012.499,-132.185,-105.823,-61.069,86.605,-61.009
C06689=1012.499,-131.955,-105.843,-59.853,86.504,-59.789
C06690=1012.499,-131.724,-105.862,-58.706,86.402,-58.639
C06691=1012.499,-131.493,-105.882,-57.623,86.298,-57.553
C06692=1012.499,-131.262,-105.901,-56.600,86.193,-56.528
C06693=1012.500,-131.030,-105.921,-55.632,86.087,-55.558
C06694=1012.499,-130.800,-105.940,-54.717,85.979,-54.641
C06695=1012.500,-130.569,-105.959,-53.852,85.871,-53.772
C06696=1012.501,-130.338,-105.980,-53.039,85.763,-52.958
C06697=1012.500,-130.107,-105.999,-52.260,85.654,-52.176
C06698=1012.501,-129.876,-106.018,-51.527,85.544,-51.441
C06699=1012.502,-129.645,-106.038,-50.823,85.432,-50.735
C06700=1012.501,-129.414,-106.057,-50.160,85.321,-50.070
C06701=1012.502,-129.183,-106.077,-49.529,85.210,-49.437
C06702=1012.503,-128.953,-106.097,-48.926,85.097,-48.834
C06703=1012.502,-128.721,-106.117,-48.352,84.984,-48.258
C06704=1012.503,-128.491,-106.136,-47.803,84.871,-47.708
C06705=1012.503,-128.260,-106.155,-47.279,84.758,-47.182
C06706=1012.503,-128.028,-106.175,-46.777,84.645,-46.678
C06707=1012.504,-127.797,-106.194,-46.297,84.530,-46.197
C06708=1012.504,-127.567,-106.214,-45.836,84.416,-45.735
C06709=1012.504,-127.336,-106.234,-45.400,84.301,-45.299
C06710=1012.505,-127.105,-106.253,-44.977,84.186,-44.874
C06711=1012.505,-126.873,-106.273,-44.575,84.071,-44.471
C06712=1012.506,-126.642,-106.292,-44.184,83.956,-44.079
C06713=1012.506,-126.412,-106.312,-43.813,83.841,-43.707
C06714=1012.506,-126.181,-106.332,-43.455,83.725,-43.350
C06715=1012.507,-125.950,-106.351,-43.111,83.610,-43.005
C06716=1012.508,-125.719,-106.370,-42.780,83.495,-42.672
C06717=1012.508,-125.487,-106.390,-42.460,83.379,-42.352
C06718=1012.509,-125.257,-106.410,-42.152,83.263,-42.044
C06719=1012.509,-125.026,-106.430,-41.858,83.147,-41.751
C06720=1012.510,-124.795,-106.449,-41.570,83.031,-41.462
C06721=1012.509,-124.564,-106.468,-41.296,82.915,-41.189
C06722=1012.510,-124.333,-106.488,-41.027,82.799,-40.920
C06723=1012.511,-124.102,-106.508,-40.771,82.683,-40.664
C06724=1012.511,-123.869,-106.527,-40.523,82.568,-40.416
C06725=1012.512,-123.639,-106.547,-40.283,82.451,-40.177
C06726=1012.512,-123.408,-106.566,-40.049,82.336,-39.943
C06727=1012.513,-123.178,-106.586,-39.827,82.221,-39.721
C06728=1012.514,-122.947,-106.606,-39.608,82.104,-39.504
C06729=1012.514,-122.716,-106.625,-39.399,81.989,-39.295
C06730=1012.515,-122.484,-106.645,-39.193,81.873,-39.090
C06731=1012.515,-122.254,-106.665,-38.995,81.758,-38.892
C06732=1012.516,-122.022,-106.685,-38.803,81.642,-38.702
C06733=1012.516,-121.791,-106.704,-38.617,81.527,-38.516
C06734=1012.517,-121.560,-106.723,-38.436,81.411,-38.338
C06735=1012.518,-121.330,-106.743,-38.260,81.296,-38.162
C06736=1012.519,-121.099,-106.763,-38.088,81.180,-37.992
C06737=1012.519,-120.867,-106.783,-37.923,81.066,-37.828
C06738=1012.520,-120.635,-106.802,-37.761,80.950,-37.668
C06739=1012.521,-120.405,-106.822,-37.606,80.835,-37.515
C06740=1012.522,-120.174,-106.842,-37.451,80.720,-37.361
C06741=1012.522,-119.942,-106.861,-37.303,80.605,-37.214
C06742=1012.523,-119.711,-106.880,-37.159,80.490,-37.072
C06743=1012.524,-119.481,-106.900,-37.018,80.376,-36.933
C06744=1012.524,-119.249,-106.920,-36.883,80.261,-36.801
C06745=1012.524,-119.018,-106.940,-36.749,80.147,-36.668
C06746=1012.526,-118.786,-106.959,-36.618,80.032,-36.540
C06747=1012.527,-118.556,-106.979,-36.492,79.918,-36.417
C06748=1012.527,-118.325,-106.999,-36.370,79.804,-36.296
C06749=1012.528,-118.094,-107.018,-36.248,79.690,-36.176
C06750=1012.529,-117.862,-107.037,-36.130,79.576,-36.062
C06751=1012.530,-117.631,-107.058,-36.016,79.462,-35.950
C06752=1012.531,-117.400,-107.077,-35.904,79.348,-35.840
C06753=1012.531,-117.169,-107.096,-35.797,79.235,-35.737
C06754=1012.531,-116.937,-107.116,-35.689,79.121,-35.631
C06755=1012.533,-116.706,-107.137,-35.586,79.008,-35.531
C06756=1012.534,-116.475,-107.156,-35.483,78.895,-35.431
C06757=1012.534,-116.244,-107.176,-35.384,78.781,-35.336
C06758=1012.535,-116.013,-107.195,-35.288,78.668,-35.243
C06759=1012.536,-115.782,-107.215,-35.192,78.556,-35.151
C06760=1012.537,-115.550,-107.235,-35.099,78.443,-35.060
C06761=1012.538,-115.319,-107.254,-35.009,78.330,-34.974
C06762=1012.539,-115.088,-107.274,-34.919,78.217,-34.887
C06763=1012.540,-114.857,-107.294,-34.833,78.105,-34.806
C06764=1012.541,-114.626,-107.313,-34.748,77.993,-34.723
C06765=1012.542,-114.394,-107.333,-34.664,77.882,-34.643
C06766=1012.543,-114.163,-107.353,-34.584,77.769,-34.567
C06767=1012.543,-113.932,-107.372,-34.504,77.658,-34.491
C06768=1012.545,-113.700,-107.392,-34.425,77.546,-34.416
C06769=1012.547,-113.279,-107.428,-34.288,77.343,-34.286
C06770=1012.548,-113.007,-107.451,-34.201,77.212,-34.204
C06771=1012.548,-112.775,-107.471,-34.129,77.101,-34.136
C06772=1012.549,-112.544,-107.491,-34.059,76.990,-34.071
C06773=1012.549,-112.312,-107.510,-33.988,76.879,-34.004
C06774=1012.551,-112.081,-107.530,-33.921,76.768,-33.941
C06775=1012.552,-111.850,-107.550,-33.854,76.658,-33.878
C06776=1012.553,-111.618,-107.569,-33.790,76.548,-33.820
C06777=1012.554,-111.387,-107.589,-33.726,76.438,-33.760
C06778=1012.555,-111.156,-107.609,-33.663,76.327,-33.702
C06779=1012.556,-110.925,-107.629,-33.602,76.217,-33.647
C06780=1012.557,-110.693,-107.648,-33.541,76.108,-33.589
C06781=1012.558,-110.462,-107.668,-33.481,75.998,-33.535
C06782=1012.559,-110.230,-107.687,-33.424,75.888,-33.483
C06783=1012.561,-109.999,-107.708,-33.367,75.779,-33.431
C06784=1012.561,-109.767,-107.727,-33.311,75.670,-33.380
C06785=1012.562,-109.536,-107.747,-33.256,75.562,-33.331
C06786=1012.563,-109.302,-107.767,-33.200,75.452,-33.280
C06787=1012.565,-109.061,-107.787,-33.145,75.339,-33.230
C06788=1012.565,-108.811,-107.808,-33.090,75.222,-33.181
C06789=1012.567,-108.551,-107.830,-33.032,75.100,-33.129
C06790=1012.568,-108.282,-107.854,-32.974,74.974,-33.079
C06791=1012.570,-108.009,-107.877,-32.916,74.847,-33.027
C06792=1012.571,-107.732,-107.899,-32.859,74.718,-32.977
C06793=1012.573,-107.456,-107.924,-32.803,74.591,-32.928
C06794=1012.574,-107.186,-107.946,-32.749,74.465,-32.881
C06795=1012.575,-106.924,-107.969,-32.697,74.343,-32.836
C06796=1012.576,-106.672,-107.991,-32.649,74.227,-32.794
C06797=1012.578,-106.429,-108.011,-32.603,74.115,-32.755
C06798=1012.579,-106.195,-108.031,-32.559,74.007,-32.717
C06799=1012.580,-105.963,-108.051,-32.516,73.900,-32.681
C06800=1012.581,-105.731,-108.071,-32.475,73.794,-32.647
C06801=1012.582,-105.500,-108.090,-32.434,73.688,-32.611
C06802=1012.583,-105.269,-108.110,-32.393,73.582,-32.577
C06803=1012.584,-105.037,-108.130,-32.354,73.476,-32.546
///RCONF 0,0,0,0,1,0,0,0,0,0,0,0,0,0,0,0,0,0,0,0,0,0,0,0
C06804=1012.586,-104.806,-108.149,-32.315,73.372,-32.512
C06805=1012.587,-104.575,-108.169,-32.276,73.266,-32.480
C06806=1012.588,-104.344,-108.188,-32.239,73.161,-32.450
C06807=1012.589,-104.114,-108.208,-32.202,73.057,-32.420
C06808=1012.590,-103.883,-108.228,-32.166,72.952,-32.392
C06809=1012.592,-103.653,-108.247,-32.130,72.848,-32.362
C06810=1012.593,-103.423,-108.267,-32.094,72.744,-32.334
C06811=1012.594,-103.193,-108.286,-32.058,72.641,-32.304
C06812=1012.596,-102.963,-108.306,-32.025,72.538,-32.278
C06813=1012.597,-102.734,-108.325,-31.991,72.435,-32.251
C06814=1012.598,-102.505,-108.345,-31.957,72.332,-32.224
C06815=1012.600,-102.276,-108.364,-31.925,72.229,-32.200
C06816=1012.601,-102.046,-108.383,-31.892,72.128,-32.174
C06817=1012.602,-101.769,-108.408,-31.854,72.004,-32.145
C06818=1012.604,-101.363,-108.442,-31.799,71.822,-32.104
C06819=1012.605,-101.135,-108.461,-31.769,71.722,-32.082
C06820=1012.606,-100.908,-108.481,-31.738,71.622,-32.057
C06821=1012.608,-100.682,-108.500,-31.710,71.522,-32.037
C06822=1012.609,-100.455,-108.519,-31.680,71.422,-32.015
C06823=1012.611,-100.229,-108.539,-31.652,71.323,-31.994
C06824=1012.612,-100.004,-108.557,-31.624,71.224,-31.974
C06825=1012.613,-99.779,-108.577,-31.597,71.125,-31.955
C06826=1012.615,-99.554,-108.596,-31.569,71.027,-31.934
C06827=1012.615,-99.330,-108.615,-31.542,70.930,-31.915
C06828=1012.617,-99.105,-108.634,-31.515,70.832,-31.896
C06829=1012.618,-98.881,-108.653,-31.489,70.735,-31.878
C06830=1012.620,-98.658,-108.672,-31.464,70.638,-31.862
C06831=1012.621,-98.434,-108.691,-31.439,70.542,-31.844
C06832=1012.622,-98.210,-108.710,-31.414,70.444,-31.827
C06833=1012.623,-97.987,-108.730,-31.389,70.348,-31.810
C06834=1012.625,-97.762,-108.748,-31.364,70.252,-31.794
C06835=1012.625,-97.540,-108.767,-31.341,70.157,-31.779
C06836=1012.627,-97.316,-108.786,-31.317,70.061,-31.763
C06837=1012.629,-97.092,-108.804,-31.293,69.966,-31.747
C06838=1012.629,-96.869,-108.824,-31.270,69.871,-31.733
C06839=1012.631,-96.644,-108.843,-31.247,69.776,-31.718
C06840=1012.632,-96.420,-108.862,-31.224,69.680,-31.704
C06841=1012.634,-96.195,-108.881,-31.202,69.586,-31.689
C06842=1012.635,-95.971,-108.900,-31.180,69.492,-31.676
C06843=1012.636,-95.746,-108.920,-31.158,69.397,-31.663
C06844=1012.638,-95.520,-108.938,-31.136,69.302,-31.649
C06845=1012.639,-95.295,-108.958,-31.114,69.208,-31.636
C06846=1012.640,-95.068,-108.977,-31.093,69.114,-31.624
C06847=1012.642,-94.842,-108.996,-31.072,69.019,-31.612
C06848=1012.644,-94.615,-109.016,-31.051,68.924,-31.600
C06849=1012.645,-94.387,-109.034,-31.031,68.830,-31.589
C06850=1012.646,-94.159,-109.054,-31.010,68.735,-31.577
C06851=1012.647,-93.930,-109.073,-30.990,68.641,-31.567
C06852=1012.649,-93.702,-109.093,-30.969,68.547,-31.554
C06853=1012.650,-93.473,-109.112,-30.950,68.453,-31.545
C06854=1012.651,-93.244,-109.131,-30.930,68.358,-31.534
C06855=1012.653,-93.013,-109.151,-30.911,68.265,-31.523
C06856=1012.654,-92.783,-109.171,-30.892,68.171,-31.515
C06857=1012.656,-92.553,-109.190,-30.873,68.077,-31.505
C06858=1012.657,-92.322,-109.210,-30.854,67.984,-31.495
C06859=1012.658,-92.091,-109.229,-30.835,67.891,-31.485
C06860=1012.660,-91.861,-109.249,-30.816,67.797,-31.476
C06861=1012.661,-91.629,-109.268,-30.798,67.705,-31.468
C06862=1012.663,-91.398,-109.288,-30.780,67.611,-31.459
C06863=1012.665,-91.166,-109.308,-30.762,67.518,-31.452
C06864=1012.665,-90.917,-109.329,-30.743,67.418,-31.442
C06865=1012.668,-90.620,-109.354,-30.720,67.300,-31.433
C06866=1012.670,-90.223,-109.388,-30.691,67.143,-31.420
C06867=1012.671,-89.946,-109.411,-30.670,67.033,-31.411
C06868=1012.673,-89.644,-109.437,-30.649,66.914,-31.403
C06869=1012.676,-89.336,-109.463,-30.627,66.792,-31.395
C06870=1012.678,-88.938,-109.497,-30.599,66.637,-31.384
C06871=1012.680,-88.539,-109.530,-30.571,66.481,-31.373
C06872=1012.682,-88.312,-109.549,-30.556,66.393,-31.368
C06873=1012.683,-88.087,-109.569,-30.541,66.306,-31.363
C06874=1012.685,-87.869,-109.587,-30.526,66.223,-31.357
C06875=1012.686,-87.655,-109.605,-30.512,66.140,-31.353
C06876=1012.688,-87.436,-109.624,-30.498,66.056,-31.348
C06877=1012.689,-87.216,-109.643,-30.484,65.971,-31.344
C06878=1012.691,-86.993,-109.662,-30.469,65.886,-31.340
C06879=1012.692,-86.763,-109.681,-30.455,65.799,-31.335
C06880=1012.692,-86.532,-109.700,-30.440,65.711,-31.330
C06881=1012.695,-86.298,-109.720,-30.426,65.622,-31.328
C06882=1012.696,-86.047,-109.741,-30.410,65.527,-31.323
C06883=1012.698,-85.777,-109.764,-30.393,65.426,-31.317
C06884=1012.699,-85.494,-109.788,-30.376,65.320,-31.313
C06885=1012.701,-85.210,-109.811,-30.359,65.213,-31.309
C06886=1012.703,-84.935,-109.836,-30.343,65.111,-31.306
C06887=1012.705,-84.679,-109.857,-30.329,65.016,-31.303
C06888=1012.706,-84.439,-109.877,-30.314,64.926,-31.299
C06889=1012.708,-84.206,-109.897,-30.301,64.841,-31.297
C06890=1012.709,-83.974,-109.917,-30.288,64.755,-31.294
C06891=1012.710,-83.741,-109.936,-30.275,64.669,-31.293
C06892=1012.712,-83.505,-109.956,-30.262,64.583,-31.290
C06893=1012.713,-83.269,-109.976,-30.249,64.497,-31.289
C06894=1012.715,-83.033,-109.996,-30.236,64.412,-31.286
C06895=1012.716,-82.798,-110.016,-30.223,64.326,-31.285
C06896=1012.718,-82.562,-110.036,-30.211,64.240,-31.283
C06897=1012.719,-82.325,-110.056,-30.198,64.155,-31.280
C06898=1012.721,-82.088,-110.076,-30.185,64.069,-31.280
C06899=1012.723,-81.851,-110.096,-30.173,63.985,-31.279
C06900=1012.724,-81.614,-110.116,-30.161,63.900,-31.277
C06901=1012.725,-81.376,-110.136,-30.149,63.815,-31.276
C06902=1012.727,-81.141,-110.156,-30.136,63.731,-31.275
C06903=1012.728,-80.905,-110.175,-30.125,63.649,-31.274
C06904=1012.730,-80.668,-110.196,-30.113,63.564,-31.274
C06905=1012.732,-80.431,-110.216,-30.101,63.481,-31.273
C06906=1012.733,-80.194,-110.236,-30.089,63.398,-31.273
C06907=1012.735,-79.955,-110.256,-30.078,63.315,-31.272
C06908=1012.736,-79.718,-110.276,-30.066,63.233,-31.272
C06909=1012.737,-79.480,-110.296,-30.055,63.150,-31.272
C06910=1012.739,-79.241,-110.316,-30.044,63.067,-31.272
C06911=1012.741,-79.003,-110.336,-30.032,62.984,-31.273
C06912=1012.742,-78.765,-110.356,-30.021,62.902,-31.273
C06913=1012.743,-78.526,-110.377,-30.010,62.821,-31.273
C06914=1012.745,-78.287,-110.397,-30.000,62.739,-31.274
C06915=1012.746,-78.049,-110.417,-29.989,62.658,-31.274
C06916=1012.748,-77.809,-110.437,-29.978,62.576,-31.275
C06917=1012.749,-77.570,-110.457,-29.967,62.495,-31.275
C06918=1012.751,-77.331,-110.477,-29.956,62.415,-31.276
C06919=1012.752,-77.092,-110.498,-29.946,62.335,-31.277
C06920=1012.754,-76.852,-110.517,-29.935,62.255,-31.278
C06921=1012.755,-76.614,-110.538,-29.925,62.174,-31.280
C06922=1012.757,-76.374,-110.557,-29.914,62.094,-31.280
C06923=1012.758,-76.134,-110.578,-29.904,62.015,-31.282
C06924=1012.760,-75.895,-110.599,-29.894,61.936,-31.284
C06925=1012.761,-75.655,-110.619,-29.884,61.857,-31.286
C06926=1012.763,-75.415,-110.638,-29.874,61.779,-31.286
C06927=1012.764,-75.175,-110.659,-29.864,61.700,-31.288
C06928=1012.766,-74.935,-110.679,-29.854,61.622,-31.289
C06929=1012.768,-74.696,-110.699,-29.844,61.545,-31.291
C06930=1012.769,-74.455,-110.719,-29.835,61.467,-31.293
C06931=1012.770,-74.215,-110.740,-29.825,61.390,-31.295
C06932=1012.771,-73.975,-110.760,-29.815,61.312,-31.297
C06933=1012.774,-73.598,-110.792,-29.800,61.192,-31.300
C06934=1012.776,-73.255,-110.821,-29.787,61.082,-31.304
C06935=1012.777,-73.014,-110.841,-29.778,61.006,-31.306
C06936=1012.779,-72.774,-110.861,-29.768,60.931,-31.308
C06937=1012.781,-72.534,-110.881,-29.760,60.856,-31.311
C06938=1012.782,-72.294,-110.901,-29.750,60.780,-31.313
C06939=1012.784,-72.053,-110.922,-29.741,60.705,-31.317
C06940=1012.785,-71.813,-110.942,-29.732,60.630,-31.319
C06941=1012.786,-71.572,-110.963,-29.723,60.556,-31.321
C06942=1012.787,-71.332,-110.983,-29.714,60.481,-31.324
C06943=1012.790,-71.091,-111.003,-29.706,60.408,-31.327
C06944=1012.791,-70.851,-111.023,-29.697,60.334,-31.330
C06945=1012.793,-70.610,-111.043,-29.689,60.261,-31.334
C06946=1012.794,-70.369,-111.063,-29.680,60.188,-31.335
C06947=1012.795,-70.128,-111.083,-29.671,60.115,-31.339
C06948=1012.796,-69.888,-111.103,-29.663,60.043,-31.342
C06949=1012.798,-69.647,-111.124,-29.654,59.971,-31.345
C06950=1012.799,-69.407,-111.144,-29.646,59.898,-31.349
C06951=1012.801,-69.166,-111.164,-29.638,59.827,-31.351
C06952=1012.802,-68.925,-111.185,-29.629,59.755,-31.354
C06953=1012.804,-68.685,-111.205,-29.621,59.684,-31.359
C06954=1012.805,-68.444,-111.225,-29.613,59.614,-31.362
C06955=1012.806,-68.203,-111.245,-29.605,59.543,-31.366
C06956=1012.808,-67.962,-111.265,-29.597,59.473,-31.369
C06957=1012.809,-67.722,-111.285,-29.589,59.403,-31.372
C06958=1012.811,-67.481,-111.306,-29.581,59.333,-31.376
C06959=1012.812,-67.241,-111.326,-29.573,59.265,-31.379
C06960=1012.813,-67.001,-111.345,-29.565,59.195,-31.383
C06961=1012.815,-66.760,-111.366,-29.558,59.127,-31.387
C06962=1012.816,-66.520,-111.386,-29.550,59.058,-31.391
C06963=1012.818,-66.280,-111.407,-29.543,58.990,-31.395
C06964=1012.819,-66.040,-111.427,-29.535,58.922,-31.399
C06965=1012.821,-65.800,-111.446,-29.527,58.855,-31.401
C06966=1012.822,-65.560,-111.467,-29.520,58.788,-31.406
C06967=1012.823,-65.320,-111.487,-29.512,58.722,-31.410
C06968=1012.825,-65.081,-111.507,-29.505,58.656,-31.414
C06969=1012.826,-64.840,-111.527,-29.498,58.589,-31.419
C06970=1012.827,-64.601,-111.547,-29.490,58.523,-31.421
C06971=1012.829,-64.362,-111.567,-29.483,58.458,-31.426
C06972=1012.829,-64.123,-111.587,-29.476,58.393,-31.430
C06973=1012.832,-63.883,-111.608,-29.469,58.328,-31.434
C06974=1012.832,-63.644,-111.627,-29.462,58.264,-31.438
C06975=1012.834,-63.405,-111.647,-29.455,58.200,-31.441
C06976=1012.835,-63.167,-111.667,-29.448,58.136,-31.446
C06977=1012.837,-62.928,-111.687,-29.441,58.072,-31.450
C06978=1012.837,-62.689,-111.708,-29.434,58.009,-31.456
C06979=1012.839,-62.451,-111.727,-29.427,57.946,-31.459
C06980=1012.840,-62.214,-111.748,-29.421,57.884,-31.463
C06981=1012.842,-61.975,-111.767,-29.414,57.822,-31.467
C06982=1012.843,-61.737,-111.787,-29.407,57.760,-31.471
C06983=1012.844,-61.500,-111.807,-29.401,57.698,-31.476
C06984=1012.846,-61.263,-111.827,-29.394,57.637,-31.481
C06985=1012.847,-61.026,-111.847,-29.388,57.577,-31.485
C06986=1012.848,-60.788,-111.867,-29.381,57.516,-31.489
C06987=1012.849,-60.552,-111.886,-29.374,57.456,-31.492
C06988=1012.851,-60.315,-111.906,-29.368,57.396,-31.497
C06989=1012.852,-60.079,-111.927,-29.362,57.336,-31.502
C06990=1012.853,-59.843,-111.946,-29.355,57.277,-31.505
C06991=1012.855,-59.606,-111.965,-29.349,57.218,-31.511
C06992=1012.856,-59.371,-111.986,-29.343,57.160,-31.515
C06993=1012.857,-59.134,-112.005,-29.337,57.102,-31.519
C06994=1012.859,-58.899,-112.025,-29.331,57.044,-31.524
C06995=1012.860,-58.664,-112.044,-29.325,56.987,-31.527
C06996=1012.861,-58.429,-112.064,-29.319,56.930,-31.532
C06997=1012.863,-58.194,-112.084,-29.313,56.873,-31.536
C06998=1012.864,-57.959,-112.104,-29.307,56.816,-31.542
C06999=1012.865,-57.724,-112.123,-29.301,56.760,-31.546
C07000=1012.865,-57.490,-112.142,-29.295,56.703,-31.550
C07001=1012.867,-57.255,-112.163,-29.289,56.649,-31.553
C07002=1012.868,-57.021,-112.182,-29.283,56.593,-31.558
C07003=1012.869,-56.787,-112.202,-29.277,56.538,-31.562
C07004=1012.870,-56.553,-112.221,-29.272,56.483,-31.568
C07005=1012.872,-56.319,-112.241,-29.266,56.429,-31.572
C07006=1012.872,-56.085,-112.260,-29.260,56.375,-31.576
C07007=1012.874,-55.851,-112.280,-29.255,56.321,-31.580
C07008=1012.875,-55.618,-112.300,-29.249,56.268,-31.585
C07009=1012.876,-55.384,-112.319,-29.244,56.214,-31.589
C07010=1012.877,-55.151,-112.338,-29.238,56.162,-31.593
C07011=1012.878,-54.917,-112.358,-29.233,56.110,-31.597
C07012=1012.880,-54.684,-112.378,-29.227,56.057,-31.603
C07013=1012.880,-54.450,-112.397,-29.222,56.004,-31.607
C07014=1012.882,-54.216,-112.417,-29.216,55.953,-31.610
C07015=1012.883,-53.982,-112.436,-29.211,55.901,-31.615
C07016=1012.885,-53.749,-112.456,-29.206,55.850,-31.620
C07017=1012.885,-53.515,-112.475,-29.200,55.799,-31.624
C07018=1012.886,-53.281,-112.495,-29.195,55.748,-31.627
C07019=1012.888,-53.048,-112.514,-29.190,55.698,-31.633
C07020=1012.889,-52.808,-112.534,-29.185,55.646,-31.636
C07021=1012.890,-52.577,-112.553,-29.180,55.597,-31.642
C07022=1012.890,-52.347,-112.573,-29.174,55.548,-31.645
C07023=1012.892,-52.113,-112.592,-29.169,55.498,-31.650
C07024=1012.893,-51.879,-112.612,-29.164,55.450,-31.654
C07025=1012.894,-51.646,-112.632,-29.159,55.400,-31.659
C07026=1012.895,-51.413,-112.651,-29.154,55.352,-31.663
C07027=1012.896,-51.179,-112.670,-29.149,55.304,-31.667
C07028=1012.897,-50.945,-112.690,-29.144,55.256,-31.671
C07029=1012.898,-50.712,-112.710,-29.139,55.207,-31.676
C07030=1012.899,-50.478,-112.729,-29.135,55.161,-31.679
C07031=1012.900,-50.245,-112.748,-29.130,55.113,-31.685
C07032=1012.901,-50.010,-112.768,-29.125,55.066,-31.687
C07033=1012.902,-49.776,-112.788,-29.120,55.019,-31.693
C07034=1012.904,-49.543,-112.807,-29.115,54.973,-31.697
C07035=1012.904,-49.309,-112.826,-29.111,54.926,-31.701
C07036=1012.905,-49.075,-112.846,-29.106,54.881,-31.706
C07037=1012.907,-48.842,-112.866,-29.101,54.836,-31.709
C07038=1012.907,-48.608,-112.885,-29.097,54.790,-31.714
C07039=1012.908,-48.374,-112.905,-29.092,54.745,-31.717
C07040=1012.910,-48.141,-112.924,-29.088,54.700,-31.722
C07041=1012.911,-47.906,-112.944,-29.083,54.655,-31.726
C07042=1012.911,-47.673,-112.964,-29.078,54.611,-31.730
C07043=1012.913,-47.439,-112.983,-29.074,54.567,-31.734
C07044=1012.913,-47.206,-113.002,-29.069,54.523,-31.738
C07045=1012.914,-46.971,-113.022,-29.065,54.480,-31.742
C07046=1012.916,-46.738,-113.041,-29.060,54.436,-31.746
C07047=1012.916,-46.505,-113.061,-29.056,54.394,-31.750
C07048=1012.917,-46.270,-113.081,-29.052,54.351,-31.754
C07049=1012.918,-46.036,-113.101,-29.047,54.309,-31.757
C07050=1012.919,-45.803,-113.119,-29.043,54.266,-31.761
C07051=1012.920,-45.569,-113.139,-29.039,54.225,-31.766
C07052=1012.921,-45.335,-113.158,-29.034,54.182,-31.769
C07053=1012.922,-45.101,-113.178,-29.030,54.141,-31.774
C07054=1012.922,-44.867,-113.198,-29.026,54.100,-31.777
C07055=1012.924,-44.633,-113.217,-29.022,54.060,-31.781
C07056=1012.925,-44.399,-113.237,-29.018,54.018,-31.786
C07057=1012.926,-44.166,-113.257,-29.014,53.978,-31.790
C07058=1012.926,-43.932,-113.276,-29.009,53.938,-31.793
C07059=1012.927,-43.698,-113.296,-29.005,53.899,-31.796
C07060=1012.929,-43.464,-113.315,-29.001,53.859,-31.800
C07061=1012.930,-43.230,-113.335,-28.997,53.819,-31.804
C07062=1012.930,-42.996,-113.354,-28.993,53.780,-31.807
C07063=1012.931,-42.762,-113.374,-28.989,53.742,-31.811
C07064=1012.931,-42.528,-113.393,-28.985,53.704,-31.814
C07065=1012.932,-42.293,-113.413,-28.981,53.665,-31.818
C07066=1012.933,-42.060,-113.433,-28.977,53.627,-31.821
C07067=1012.934,-41.826,-113.451,-28.974,53.590,-31.826
C07068=1012.935,-41.593,-113.471,-28.970,53.552,-31.830
C07069=1012.936,-41.358,-113.491,-28.966,53.515,-31.832
C07070=1012.937,-41.124,-113.510,-28.962,53.478,-31.835
C07071=1012.938,-40.890,-113.530,-28.959,53.441,-31.840
C07072=1012.938,-40.656,-113.549,-28.955,53.405,-31.843
C07073=1012.939,-40.422,-113.569,-28.951,53.369,-31.847
C07074=1012.940,-40.188,-113.589,-28.947,53.332,-31.850
C07075=1012.941,-39.953,-113.608,-28.944,53.297,-31.853
C07076=1012.941,-39.720,-113.628,-28.940,53.261,-31.856
C07077=1012.942,-39.486,-113.647,-28.937,53.227,-31.860
C07078=1012.943,-39.251,-113.667,-28.933,53.191,-31.863
C07079=1012.944,-39.017,-113.687,-28.929,53.157,-31.867
C07080=1012.944,-38.783,-113.706,-28.926,53.123,-31.870
C07081=1012.945,-38.549,-113.725,-28.922,53.089,-31.873
C07082=1012.946,-38.314,-113.745,-28.919,53.055,-31.877
C07083=1012.947,-38.081,-113.765,-28.915,53.021,-31.878
C07084=1012.947,-37.847,-113.784,-28.912,52.988,-31.882
C07085=1012.948,-37.613,-113.803,-28.908,52.955,-31.884
C07086=1012.949,-37.378,-113.824,-28.905,52.921,-31.889
C07087=1012.950,-37.144,-113.843,-28.902,52.889,-31.891
C07088=1012.950,-36.910,-113.862,-28.899,52.857,-31.895
C07089=1012.951,-36.676,-113.881,-28.895,52.825,-31.897
C07090=1012.952,-36.442,-113.902,-28.892,52.794,-31.900
C07091=1012.953,-36.208,-113.921,-28.889,52.762,-31.903
C07092=1012.953,-35.973,-113.940,-28.885,52.730,-31.907
C07093=1012.954,-35.739,-113.960,-28.882,52.700,-31.909
C07094=1012.955,-35.505,-113.980,-28.879,52.669,-31.911
C07095=1012.955,-35.271,-113.999,-28.876,52.639,-31.914
C07096=1012.956,-35.037,-114.018,-28.872,52.608,-31.916
C07097=1012.957,-34.803,-114.038,-28.869,52.578,-31.919
C07098=1012.958,-34.568,-114.058,-28.866,52.548,-31.922
C07099=1012.958,-34.334,-114.078,-28.863,52.519,-31.926
C07100=1012.958,-34.100,-114.097,-28.860,52.489,-31.927
C07101=1012.959,-33.866,-114.117,-28.857,52.460,-31.931
C07102=1012.960,-33.632,-114.136,-28.854,52.431,-31.932
C07103=1012.960,-33.397,-114.156,-28.851,52.403,-31.935
C07104=1012.961,-33.163,-114.175,-28.848,52.374,-31.937
C07105=1012.961,-32.929,-114.194,-28.845,52.347,-31.940
C07106=1012.963,-32.695,-114.214,-28.842,52.318,-31.943
C07107=1012.963,-32.460,-114.234,-28.840,52.292,-31.944
C07108=1012.963,-32.226,-114.253,-28.837,52.264,-31.947
C07109=1012.964,-31.992,-114.273,-28.834,52.238,-31.949
C07110=1012.964,-31.759,-114.293,-28.831,52.210,-31.952
C07111=1012.966,-31.524,-114.312,-28.828,52.183,-31.954
C07112=1012.966,-31.290,-114.332,-28.826,52.157,-31.957
C07113=1012.966,-31.055,-114.351,-28.823,52.132,-31.957
C07114=1012.967,-30.822,-114.371,-28.820,52.106,-31.960
C07115=1012.967,-30.588,-114.391,-28.817,52.080,-31.962
C07116=1012.968,-30.353,-114.410,-28.815,52.055,-31.963
C07117=1012.969,-30.119,-114.429,-28.812,52.030,-31.967
C07118=1012.969,-29.884,-114.449,-28.809,52.005,-31.968
C07119=1012.969,-29.651,-114.469,-28.807,51.981,-31.970
C07120=1012.970,-29.416,-114.488,-28.804,51.956,-31.972
C07121=1012.970,-29.182,-114.508,-28.802,51.932,-31.974
C07122=1012.971,-28.948,-114.527,-28.799,51.908,-31.976
C07123=1012.972,-28.713,-114.546,-28.797,51.886,-31.977
C07124=1012.972,-28.480,-114.567,-28.794,51.862,-31.980
C07125=1012.972,-28.245,-114.586,-28.792,51.839,-31.980
C07126=1012.973,-28.011,-114.605,-28.789,51.815,-31.983
C07127=1012.973,-27.777,-114.625,-28.787,51.793,-31.984
C07128=1012.974,-27.543,-114.645,-28.785,51.771,-31.986
C07129=1012.974,-27.309,-114.665,-28.782,51.749,-31.988
C07130=1012.975,-27.075,-114.684,-28.780,51.727,-31.990
C07131=1012.975,-26.841,-114.703,-28.777,51.706,-31.990
C07132=1012.975,-26.607,-114.724,-28.775,51.684,-31.993
C07133=1012.976,-26.373,-114.743,-28.773,51.664,-31.993
C07134=1012.977,-26.138,-114.762,-28.770,51.643,-31.994
C07135=1012.977,-25.904,-114.782,-28.768,51.622,-31.997
C07136=1012.977,-25.670,-114.802,-28.766,51.601,-31.998
C07137=1012.978,-25.436,-114.821,-28.764,51.581,-31.999
C07138=1012.978,-25.202,-114.841,-28.762,51.562,-31.999
C07139=1012.979,-24.968,-114.860,-28.759,51.542,-32.001
C07140=1012.979,-24.733,-114.880,-28.758,51.523,-32.003
